C05360=1017.333,121.413,-117.741,166.979,53.925,159.921
C05361=1017.328,121.164,-117.723,166.976,53.934,159.922
C05362=1017.323,120.915,-117.704,166.972,53.942,159.923
C05363=1017.318,120.666,-117.685,166.969,53.951,159.924
C05364=1017.314,120.417,-117.667,166.966,53.960,159.926
C05365=1017.309,120.168,-117.648,166.963,53.969,159.927
C05366=1017.303,119.918,-117.630,166.960,53.978,159.928
C05367=1017.298,119.669,-117.612,166.957,53.987,159.929
C05368=1017.293,119.420,-117.593,166.954,53.996,159.930
C05369=1017.288,119.170,-117.575,166.951,54.005,159.931
C05370=1017.284,118.921,-117.557,166.948,54.014,159.932
C05371=1017.279,118.672,-117.538,166.945,54.023,159.934
C05372=1017.274,118.423,-117.520,166.942,54.031,159.934
C05373=1017.269,118.174,-117.501,166.939,54.040,159.936
C05374=1017.264,117.924,-117.483,166.937,54.049,159.937
C05375=1017.260,117.675,-117.465,166.934,54.058,159.938
C05376=1017.254,117.426,-117.446,166.931,54.067,159.939
C05377=1017.249,117.176,-117.428,166.928,54.076,159.940
C05378=1017.244,116.927,-117.409,166.925,54.085,159.941
C05379=1017.240,116.677,-117.391,166.922,54.094,159.943
C05380=1017.235,116.428,-117.373,166.919,54.103,159.944
C05381=1017.230,116.179,-117.354,166.916,54.111,159.945
C05382=1017.226,115.930,-117.335,166.913,54.120,159.946
C05383=1017.221,115.680,-117.317,166.911,54.129,159.947
C05384=1017.216,115.431,-117.299,166.907,54.137,159.948
C05385=1017.211,115.182,-117.281,166.904,54.147,159.949
C05386=1017.206,114.933,-117.262,166.902,54.156,159.950
C05387=1017.201,114.684,-117.244,166.899,54.165,159.952
C05388=1017.197,114.434,-117.226,166.895,54.173,159.953
C05389=1017.192,114.185,-117.208,166.892,54.182,159.954
C05390=1017.187,113.936,-117.189,166.890,54.191,159.955
C05391=1017.182,113.686,-117.171,166.887,54.199,159.956
C05392=1017.177,113.437,-117.153,166.884,54.208,159.957
C05393=1017.172,113.188,-117.134,166.881,54.218,159.958
C05394=1017.168,112.939,-117.116,166.878,54.227,159.960
C05395=1017.163,112.689,-117.098,166.875,54.235,159.960
C05396=1017.158,112.440,-117.080,166.873,54.244,159.962
C05397=1017.153,112.191,-117.062,166.870,54.253,159.963
C05398=1017.148,111.941,-117.043,166.867,54.261,159.964
C05399=1017.144,111.692,-117.025,166.864,54.270,159.965
C05400=1017.138,111.443,-117.008,166.861,54.280,159.966
C05401=1017.133,111.194,-116.990,166.858,54.289,159.967
C05402=1017.129,110.944,-116.971,166.855,54.298,159.969
C05403=1017.124,110.695,-116.953,166.852,54.307,159.970
C05404=1017.118,110.446,-116.936,166.849,54.315,159.971
C05405=1017.114,110.196,-116.918,166.846,54.324,159.972
C05406=1017.109,109.947,-116.900,166.843,54.334,159.973
C05407=1017.104,109.698,-116.883,166.842,54.342,159.974
C05408=1017.099,109.448,-116.864,166.839,54.351,159.976
C05409=1017.094,109.199,-116.846,166.835,54.360,159.977
C05410=1017.088,108.950,-116.829,166.832,54.369,159.978
C05411=1017.084,108.700,-116.810,166.830,54.378,159.979
C05412=1017.079,108.450,-116.793,166.827,54.387,159.980
C05413=1017.074,108.201,-116.775,166.824,54.396,159.981
C05414=1017.069,107.952,-116.757,166.821,54.406,159.982
C05415=1017.063,107.703,-116.740,166.818,54.415,159.984
C05416=1017.059,107.453,-116.722,166.815,54.424,159.985
C05417=1017.053,107.172,-116.702,166.812,54.434,159.986
C05418=1017.047,106.890,-116.682,166.808,54.444,159.987
C05419=1017.042,106.608,-116.662,166.805,54.455,159.989
C05420=1017.035,106.327,-116.642,166.803,54.464,159.990
C05421=1017.032,106.078,-116.625,166.800,54.474,159.991
C05422=1017.026,105.829,-116.607,166.797,54.483,159.993
C05423=1017.021,105.579,-116.589,166.794,54.491,159.993
C05424=1017.016,105.330,-116.572,166.791,54.500,159.995
C05425=1017.011,105.080,-116.554,166.788,54.509,159.996
C05426=1017.006,104.831,-116.537,166.785,54.519,159.997
C05427=1017.001,104.582,-116.518,166.782,54.528,159.998
C05428=1016.997,104.332,-116.501,166.780,54.537,159.999
C05429=1016.991,104.083,-116.483,166.776,54.545,160.000
C05430=1016.986,103.833,-116.465,166.773,54.555,160.002
C05431=1016.982,103.585,-116.449,166.772,54.563,160.003
C05432=1016.977,103.335,-116.431,166.769,54.573,160.004
C05433=1016.971,103.086,-116.413,166.766,54.582,160.005
C05434=1016.967,102.836,-116.396,166.763,54.591,160.006
C05435=1016.961,102.587,-116.378,166.760,54.599,160.007
C05436=1016.957,102.338,-116.360,166.757,54.608,160.009
C05437=1016.951,102.088,-116.343,166.754,54.618,160.010
C05438=1016.947,101.839,-116.325,166.751,54.627,160.011
C05439=1016.942,101.590,-116.308,166.749,54.635,160.012
C05440=1016.937,101.340,-116.290,166.746,54.644,160.013
C05441=1016.932,101.091,-116.272,166.744,54.653,160.014
C05442=1016.927,100.841,-116.255,166.741,54.662,160.016
C05443=1016.922,100.592,-116.237,166.738,54.672,160.017
C05444=1016.917,100.343,-116.220,166.735,54.680,160.018
C05445=1016.913,100.094,-116.202,166.732,54.689,160.019
C05446=1016.907,99.845,-116.185,166.730,54.698,160.020
C05447=1016.903,99.595,-116.167,166.727,54.707,160.021
C05448=1016.897,99.346,-116.150,166.724,54.716,160.022
C05449=1016.893,99.096,-116.132,166.721,54.725,160.024
C05450=1016.887,98.847,-116.115,166.718,54.734,160.025
C05451=1016.883,98.598,-116.098,166.716,54.743,160.026
C05452=1016.878,98.348,-116.080,166.713,54.752,160.027
C05453=1016.873,98.099,-116.063,166.710,54.761,160.028
C05454=1016.868,97.849,-116.046,166.707,54.770,160.029
C05455=1016.862,97.600,-116.029,166.704,54.779,160.031
C05456=1016.858,97.351,-116.012,166.701,54.789,160.032
C05457=1016.853,97.102,-115.994,166.700,54.797,160.033
C05458=1016.848,96.852,-115.977,166.697,54.807,160.034
C05459=1016.842,96.602,-115.961,166.694,54.816,160.035
C05460=1016.838,96.353,-115.942,166.691,54.825,160.037
C05461=1016.833,96.104,-115.926,166.688,54.833,160.038
C05462=1016.828,95.854,-115.909,166.685,54.843,160.039
C05463=1016.822,95.605,-115.892,166.683,54.852,160.040
C05464=1016.817,95.356,-115.875,166.680,54.861,160.041
C05465=1016.813,95.106,-115.858,166.677,54.870,160.042
C05466=1016.808,94.857,-115.840,166.674,54.880,160.044
C05467=1016.802,94.608,-115.823,166.671,54.888,160.045
C05468=1016.797,94.358,-115.806,166.669,54.897,160.046
C05469=1016.793,94.109,-115.789,166.667,54.906,160.047
C05470=1016.788,93.860,-115.772,166.664,54.915,160.048
C05471=1016.783,93.610,-115.755,166.661,54.925,160.050
C05472=1016.777,93.361,-115.737,166.658,54.933,160.050
C05473=1016.773,93.112,-115.720,166.655,54.942,160.052
C05474=1016.768,92.862,-115.703,166.652,54.951,160.053
C05475=1016.763,92.613,-115.686,166.650,54.961,160.054
C05476=1016.758,92.364,-115.669,166.647,54.970,160.055
C05477=1016.753,92.115,-115.652,166.645,54.978,160.056
C05478=1016.748,91.865,-115.635,166.642,54.987,160.058
C05479=1016.743,91.615,-115.618,166.639,54.997,160.059
C05480=1016.738,91.367,-115.601,166.637,55.006,160.060
C05481=1016.732,91.085,-115.582,166.633,55.015,160.061
C05482=1016.727,90.803,-115.562,166.631,55.025,160.063
C05483=1016.722,90.522,-115.543,166.627,55.036,160.064
C05484=1016.716,90.240,-115.524,166.624,55.046,160.065
C05485=1016.711,89.991,-115.507,166.621,55.055,160.066
C05486=1016.706,89.742,-115.490,166.619,55.063,160.067
C05487=1016.701,89.492,-115.473,166.616,55.073,160.069
C05488=1016.696,89.243,-115.456,166.614,55.082,160.070
C05489=1016.692,88.994,-115.439,166.611,55.091,160.071
C05490=1016.686,88.744,-115.422,166.608,55.100,160.072
C05491=1016.681,88.494,-115.406,166.605,55.109,160.073
C05492=1016.676,88.245,-115.389,166.602,55.118,160.074
C05493=1016.671,87.996,-115.372,166.600,55.127,160.076
C05494=1016.666,87.746,-115.355,166.597,55.137,160.077
C05495=1016.661,87.497,-115.339,166.594,55.146,160.078
C05496=1016.656,87.247,-115.322,166.593,55.155,160.079
C05497=1016.651,86.998,-115.305,166.590,55.163,160.080
C05498=1016.646,86.749,-115.289,166.587,55.173,160.082
C05499=1016.640,86.500,-115.272,166.584,55.182,160.083
C05500=1016.635,86.250,-115.256,166.581,55.191,160.084
C05501=1016.631,86.001,-115.239,166.579,55.200,160.085
C05502=1016.625,85.751,-115.222,166.576,55.210,160.086
C05503=1016.620,85.502,-115.205,166.573,55.218,160.087
C05504=1016.616,85.253,-115.189,166.570,55.228,160.089
C05505=1016.610,85.003,-115.172,166.568,55.237,160.090
C05506=1016.606,84.754,-115.156,166.565,55.246,160.091
C05507=1016.601,84.504,-115.139,166.562,55.255,160.092
C05508=1016.595,84.255,-115.122,166.560,55.263,160.093
C05509=1016.590,84.006,-115.106,166.557,55.273,160.095
C05510=1016.585,83.756,-115.089,166.555,55.282,160.096
C05511=1016.580,83.507,-115.073,166.552,55.291,160.097
C05512=1016.575,83.257,-115.057,166.550,55.301,160.098
C05513=1016.570,83.007,-115.040,166.546,55.309,160.099
C05514=1016.565,82.759,-115.023,166.544,55.318,160.100
C05515=1016.560,82.509,-115.006,166.541,55.328,160.102
C05516=1016.556,82.260,-114.990,166.539,55.337,160.103
C05517=1016.550,82.010,-114.973,166.536,55.345,160.104
C05518=1016.546,81.761,-114.957,166.534,55.354,160.105
C05519=1016.540,81.512,-114.940,166.531,55.364,160.106
C05520=1016.535,81.262,-114.923,166.528,55.372,160.107
C05521=1016.530,81.013,-114.908,166.525,55.382,160.109
C05522=1016.525,80.763,-114.891,166.523,55.391,160.110
C05523=1016.521,80.514,-114.874,166.521,55.400,160.111
C05524=1016.515,80.264,-114.857,166.518,55.408,160.112
C05525=1016.511,80.015,-114.841,166.515,55.418,160.113
C05526=1016.506,79.766,-114.824,166.513,55.427,160.115
C05527=1016.501,79.516,-114.808,166.509,55.436,160.116
C05528=1016.496,79.267,-114.792,166.507,55.445,160.117
C05529=1016.491,79.018,-114.776,166.505,55.454,160.118
C05530=1016.485,78.768,-114.759,166.502,55.462,160.119
C05531=1016.481,78.519,-114.742,166.499,55.472,160.120
C05532=1016.476,78.269,-114.726,166.497,55.481,160.122
C05533=1016.471,78.020,-114.710,166.494,55.490,160.123
C05534=1016.466,77.770,-114.693,166.492,55.499,160.124
C05535=1016.461,77.521,-114.676,166.489,55.507,160.125
C05536=1016.456,77.272,-114.659,166.486,55.516,160.126
C05537=1016.452,77.022,-114.644,166.484,55.526,160.127
C05538=1016.446,76.773,-114.627,166.481,55.534,160.128
C05539=1016.441,76.524,-114.611,166.478,55.544,160.130
C05540=1016.436,76.274,-114.595,166.477,55.553,160.131
C05541=1016.432,76.025,-114.578,166.474,55.562,160.132
C05542=1016.426,75.775,-114.562,166.471,55.570,160.133
C05543=1016.422,75.526,-114.546,166.468,55.580,160.134
C05544=1016.416,75.276,-114.530,166.466,55.589,160.136
C05545=1016.411,74.995,-114.512,166.463,55.600,160.137
C05546=1016.404,74.713,-114.494,166.460,55.610,160.138
C05547=1016.399,74.432,-114.475,166.457,55.619,160.139
C05548=1016.393,74.151,-114.457,166.454,55.630,160.141
C05549=1016.388,73.901,-114.441,166.451,55.639,160.142
C05550=1016.383,73.652,-114.425,166.449,55.649,160.143
C05551=1016.378,73.402,-114.409,166.445,55.657,160.144
C05552=1016.373,73.153,-114.393,166.444,55.666,160.146
C05553=1016.368,72.904,-114.377,166.441,55.675,160.147
C05554=1016.363,72.654,-114.361,166.438,55.684,160.148
C05555=1016.358,72.405,-114.345,166.436,55.693,160.149
C05556=1016.353,72.155,-114.329,166.433,55.703,160.150
C05557=1016.348,71.906,-114.312,166.430,55.711,160.151
C05558=1016.343,71.656,-114.297,166.428,55.721,160.152
C05559=1016.338,71.407,-114.280,166.426,55.730,160.154
C05560=1016.333,71.158,-114.265,166.423,55.738,160.155
C05561=1016.328,70.908,-114.248,166.420,55.748,160.156
C05562=1016.323,70.659,-114.232,166.418,55.757,160.157
C05563=1016.318,70.409,-114.216,166.415,55.766,160.158
C05564=1016.313,70.160,-114.200,166.412,55.775,160.159
C05565=1016.308,69.911,-114.185,166.411,55.784,160.161
C05566=1016.303,69.661,-114.168,166.408,55.793,160.162
C05567=1016.298,69.412,-114.153,166.405,55.802,160.163
C05568=1016.293,69.162,-114.136,166.403,55.811,160.164
C05569=1016.288,68.912,-114.120,166.399,55.820,160.165
C05570=1016.283,68.664,-114.104,166.397,55.829,160.167
C05571=1016.278,68.414,-114.088,166.395,55.837,160.168
C05572=1016.273,68.164,-114.073,166.392,55.847,160.169
C05573=1016.269,67.915,-114.057,166.390,55.856,160.170
C05574=1016.263,67.665,-114.041,166.387,55.865,160.171
C05575=1016.259,67.416,-114.025,166.384,55.874,160.172
C05576=1016.253,67.167,-114.009,166.382,55.884,160.174
C05577=1016.248,66.917,-113.994,166.380,55.892,160.175
C05578=1016.243,66.668,-113.978,166.377,55.901,160.176
C05579=1016.237,66.418,-113.962,166.375,55.911,160.177
C05580=1016.233,66.169,-113.946,166.372,55.919,160.178
C05581=1016.228,65.919,-113.931,166.369,55.929,160.179
C05582=1016.222,65.670,-113.915,166.367,55.938,160.181
C05583=1016.218,65.420,-113.899,166.364,55.947,160.182
C05584=1016.213,65.171,-113.884,166.362,55.956,160.183
C05585=1016.208,64.921,-113.868,166.359,55.964,160.184
C05586=1016.202,64.672,-113.852,166.357,55.974,160.185
C05587=1016.197,64.423,-113.837,166.354,55.983,160.187
C05588=1016.192,64.173,-113.820,166.351,55.992,160.188
C05589=1016.187,63.923,-113.805,166.349,56.001,160.189
C05590=1016.182,63.674,-113.790,166.346,56.011,160.190
C05591=1016.178,63.425,-113.774,166.344,56.019,160.191
C05592=1016.172,63.175,-113.758,166.342,56.028,160.192
C05593=1016.167,62.926,-113.743,166.339,56.037,160.193
C05594=1016.163,62.676,-113.727,166.336,56.046,160.195
C05595=1016.157,62.426,-113.712,166.334,56.056,160.196
C05596=1016.152,62.177,-113.696,166.331,56.064,160.197
C05597=1016.147,61.928,-113.681,166.328,56.074,160.198
C05598=1016.141,61.678,-113.666,166.326,56.083,160.199
C05599=1016.136,61.429,-113.651,166.323,56.093,160.201
C05600=1016.131,61.179,-113.635,166.320,56.101,160.202
C05601=1016.126,60.930,-113.620,166.318,56.111,160.203
C05602=1016.121,60.680,-113.605,166.316,56.120,160.204
C05603=1016.116,60.431,-113.589,166.314,56.129,160.206
C05604=1016.111,60.182,-113.574,166.311,56.138,160.206
C05605=1016.105,59.932,-113.559,166.308,56.147,160.208
C05606=1016.100,59.682,-113.544,166.306,56.157,160.209
C05607=1016.096,59.433,-113.528,166.303,56.166,160.210
C05608=1016.090,59.184,-113.513,166.300,56.175,160.211
C05609=1016.084,58.903,-113.496,166.298,56.185,160.213
C05610=1016.079,58.621,-113.479,166.295,56.196,160.214
C05611=1016.073,58.340,-113.461,166.293,56.206,160.215
C05612=1016.067,58.058,-113.444,166.289,56.216,160.217
C05613=1016.062,57.808,-113.429,166.287,56.225,160.218
C05614=1016.057,57.559,-113.413,166.284,56.235,160.219
C05615=1016.052,57.310,-113.398,166.281,56.243,160.220
C05616=1016.047,57.060,-113.383,166.279,56.253,160.221
C05617=1016.042,56.811,-113.368,166.276,56.262,160.223
C05618=1016.036,56.561,-113.352,166.273,56.271,160.224
C05619=1016.031,56.312,-113.337,166.272,56.280,160.225
C05620=1016.026,56.063,-113.322,166.269,56.289,160.226
C05621=1016.021,55.813,-113.307,166.267,56.298,160.227
C05622=1016.016,55.563,-113.292,166.264,56.307,160.228
C05623=1016.010,55.314,-113.277,166.261,56.316,160.229
C05624=1016.005,55.064,-113.262,166.259,56.326,160.231
C05625=1016.000,54.815,-113.246,166.256,56.334,160.232
C05626=1015.995,54.566,-113.231,166.253,56.344,160.233
C05627=1015.990,54.316,-113.216,166.252,56.352,160.234
C05628=1015.985,54.067,-113.201,166.249,56.361,160.235
C05629=1015.980,53.817,-113.186,166.246,56.370,160.236
C05630=1015.975,53.567,-113.171,166.244,56.380,160.238
C05631=1015.970,53.318,-113.156,166.241,56.388,160.239
C05632=1015.965,53.069,-113.141,166.238,56.398,160.240
C05633=1015.960,52.820,-113.125,166.237,56.406,160.241
C05634=1015.955,52.570,-113.110,166.234,56.416,160.242
C05635=1015.950,52.320,-113.096,166.231,56.424,160.243
C05636=1015.945,52.070,-113.080,166.229,56.434,160.245
C05637=1015.940,51.821,-113.064,166.226,56.442,160.246
C05638=1015.935,51.572,-113.049,166.225,56.452,160.247
C05639=1015.930,51.322,-113.034,166.222,56.460,160.248
C05640=1015.925,51.072,-113.020,166.219,56.470,160.249
C05641=1015.920,50.823,-113.004,166.216,56.478,160.250
C05642=1015.915,50.574,-112.989,166.214,56.488,160.252
C05643=1015.910,50.325,-112.974,166.212,56.496,160.253
C05644=1015.905,50.074,-112.959,166.209,56.505,160.254
C05645=1015.900,49.825,-112.944,166.207,56.514,160.255
C05646=1015.895,49.575,-112.929,166.204,56.523,160.256
C05647=1015.889,49.326,-112.914,166.201,56.533,160.257
C05648=1015.885,49.076,-112.899,166.200,56.541,160.258
C05649=1015.880,48.827,-112.884,166.197,56.550,160.259
C05650=1015.875,48.578,-112.869,166.194,56.559,160.261
C05651=1015.870,48.329,-112.854,166.191,56.568,160.262
C05652=1015.865,48.079,-112.839,166.189,56.576,160.263
C05653=1015.860,47.829,-112.824,166.187,56.586,160.264
C05654=1015.855,47.580,-112.809,166.184,56.594,160.265
C05655=1015.850,47.331,-112.794,166.181,56.603,160.266
C05656=1015.845,47.081,-112.779,166.180,56.612,160.268
C05657=1015.839,46.831,-112.764,166.177,56.621,160.268
C05658=1015.834,46.582,-112.749,166.174,56.630,160.269
C05659=1015.830,46.332,-112.734,166.171,56.639,160.270
C05660=1015.825,46.083,-112.719,166.170,56.648,160.272
C05661=1015.819,45.833,-112.704,166.167,56.656,160.273
C05662=1015.815,45.583,-112.689,166.164,56.665,160.274
C05663=1015.810,45.334,-112.674,166.163,56.674,160.275
C05664=1015.805,45.085,-112.659,166.160,56.683,160.276
C05665=1015.800,44.835,-112.645,166.157,56.692,160.277
C05666=1015.795,44.586,-112.629,166.154,56.701,160.278
C05667=1015.790,44.336,-112.614,166.152,56.709,160.280
C05668=1015.785,44.087,-112.600,166.150,56.718,160.281
C05669=1015.780,43.837,-112.585,166.147,56.727,160.282
C05670=1015.775,43.587,-112.570,166.145,56.736,160.283
C05671=1015.770,43.338,-112.555,166.143,56.744,160.284
C05672=1015.765,43.089,-112.540,166.140,56.753,160.285
C05673=1015.760,42.831,-112.524,166.138,56.762,160.286
C05674=1015.755,42.574,-112.509,166.135,56.771,160.287
C05675=1015.751,42.315,-112.494,166.133,56.780,160.289
C05676=1015.745,42.058,-112.479,166.130,56.789,160.290
C05677=1015.740,41.809,-112.464,166.127,56.798,160.291
C05678=1015.735,41.559,-112.449,166.125,56.807,160.292
C05679=1015.730,41.310,-112.435,166.122,56.816,160.293
C05680=1015.725,41.060,-112.420,166.120,56.825,160.294
C05681=1015.720,40.810,-112.406,166.118,56.834,160.295
C05682=1015.715,40.561,-112.390,166.115,56.843,160.296
C05683=1015.710,40.311,-112.377,166.112,56.852,160.297
C05684=1015.705,40.062,-112.361,166.111,56.861,160.299
C05685=1015.701,39.813,-112.347,166.108,56.870,160.300
C05686=1015.695,39.563,-112.333,166.105,56.878,160.301
C05687=1015.690,39.314,-112.318,166.103,56.887,160.302
C05688=1015.685,39.064,-112.304,166.101,56.896,160.303
C05689=1015.680,38.815,-112.289,166.099,56.905,160.304
C05690=1015.675,38.565,-112.275,166.096,56.914,160.305
C05691=1015.670,38.315,-112.260,166.093,56.923,160.306
C05692=1015.665,38.066,-112.245,166.092,56.932,160.308
C05693=1015.660,37.816,-112.231,166.089,56.941,160.309
C05694=1015.655,37.567,-112.217,166.086,56.949,160.310
C05695=1015.650,37.317,-112.202,166.083,56.958,160.311
C05696=1015.645,37.068,-112.187,166.081,56.967,160.312
C05697=1015.639,36.818,-112.173,166.079,56.976,160.313
C05698=1015.635,36.568,-112.159,166.076,56.985,160.314
C05699=1015.630,36.319,-112.144,166.074,56.993,160.316
C05700=1015.625,36.070,-112.130,166.072,57.002,160.317
C05701=1015.620,35.820,-112.116,166.069,57.012,160.318
C05702=1015.615,35.571,-112.102,166.067,57.020,160.319
C05703=1015.610,35.321,-112.087,166.064,57.029,160.320
C05704=1015.604,35.072,-112.073,166.061,57.038,160.321
C05705=1015.599,34.822,-112.058,166.060,57.047,160.322
C05706=1015.594,34.572,-112.044,166.057,57.056,160.323
C05707=1015.589,34.322,-112.030,166.054,57.065,160.324
C05708=1015.584,34.073,-112.017,166.051,57.074,160.325
C05709=1015.580,33.824,-112.002,166.049,57.083,160.327
C05710=1015.574,33.574,-111.988,166.047,57.092,160.328
C05711=1015.569,33.325,-111.973,166.044,57.100,160.329
C05712=1015.564,33.075,-111.959,166.042,57.109,160.330
C05713=1015.558,32.826,-111.945,166.039,57.119,160.331
C05714=1015.553,32.576,-111.931,166.038,57.127,160.332
C05715=1015.548,32.327,-111.917,166.035,57.136,160.333
C05716=1015.544,32.077,-111.903,166.032,57.145,160.334
C05717=1015.538,31.827,-111.889,166.029,57.154,160.335
C05718=1015.533,31.577,-111.875,166.028,57.163,160.337
C05719=1015.528,31.328,-111.861,166.025,57.172,160.338
C05720=1015.523,31.078,-111.846,166.023,57.181,160.339
C05721=1015.518,30.829,-111.833,166.020,57.189,160.340
C05722=1015.513,30.580,-111.818,166.018,57.198,160.341
C05723=1015.508,30.330,-111.804,166.015,57.207,160.342
C05724=1015.503,30.080,-111.789,166.012,57.215,160.343
C05725=1015.498,29.807,-111.774,166.010,57.225,160.345
C05726=1015.492,29.534,-111.759,166.007,57.235,160.346
C05727=1015.487,29.260,-111.744,166.005,57.245,160.347
C05728=1015.481,28.987,-111.729,166.003,57.254,160.348
C05729=1015.476,28.737,-111.714,166.000,57.263,160.349
C05730=1015.471,28.488,-111.701,165.997,57.272,160.350
C05731=1015.467,28.238,-111.686,165.995,57.280,160.352
C05732=1015.461,27.989,-111.672,165.993,57.289,160.353
C05733=1015.456,27.739,-111.658,165.990,57.298,160.354
C05734=1015.451,27.490,-111.644,165.988,57.306,160.355
C05735=1015.446,27.240,-111.630,165.985,57.315,160.356
C05736=1015.441,26.990,-111.616,165.983,57.324,160.357
C05737=1015.436,26.710,-111.600,165.980,57.334,160.358
C05738=1015.429,26.428,-111.585,165.977,57.344,160.359
C05739=1015.423,26.147,-111.569,165.975,57.355,160.361
C05740=1015.418,25.866,-111.554,165.972,57.364,160.362
C05741=1015.413,25.616,-111.540,165.970,57.373,160.363
C05742=1015.408,25.366,-111.525,165.967,57.382,160.364
C05743=1015.403,25.116,-111.512,165.965,57.390,160.365
C05744=1015.398,24.867,-111.499,165.962,57.399,160.366
C05745=1015.392,24.618,-111.485,165.960,57.408,160.367
C05746=1015.388,24.368,-111.470,165.957,57.417,160.368
C05747=1015.383,24.119,-111.457,165.955,57.425,160.369
C05748=1015.378,23.869,-111.444,165.953,57.434,160.370
C05749=1015.372,23.619,-111.430,165.950,57.443,160.371
C05750=1015.367,23.370,-111.416,165.947,57.452,160.373
C05751=1015.363,23.120,-111.402,165.945,57.460,160.374
C05752=1015.357,22.871,-111.388,165.943,57.469,160.375
C05753=1015.352,22.621,-111.375,165.940,57.478,160.376
C05754=1015.347,22.372,-111.361,165.938,57.487,160.377
C05755=1015.342,22.122,-111.348,165.935,57.495,160.378
C05756=1015.337,21.872,-111.334,165.933,57.504,160.379
C05757=1015.332,21.623,-111.320,165.930,57.513,160.380
C05758=1015.327,21.373,-111.307,165.928,57.522,160.381
C05759=1015.321,21.124,-111.293,165.926,57.531,160.382
C05760=1015.317,20.874,-111.280,165.923,57.539,160.383
C05761=1015.312,20.624,-111.265,165.921,57.548,160.385
C05762=1015.307,20.375,-111.252,165.919,57.557,160.386
C05763=1015.302,20.125,-111.239,165.916,57.566,160.387
C05764=1015.297,19.876,-111.225,165.914,57.574,160.388
C05765=1015.291,19.626,-111.211,165.912,57.583,160.389
C05766=1015.287,19.377,-111.197,165.908,57.591,160.390
C05767=1015.282,19.127,-111.184,165.907,57.600,160.391
C05768=1015.277,18.878,-111.170,165.904,57.609,160.392
C05769=1015.272,18.628,-111.157,165.901,57.617,160.393
C05770=1015.266,18.378,-111.143,165.900,57.626,160.394
C05771=1015.261,18.129,-111.130,165.897,57.635,160.395
C05772=1015.256,17.879,-111.117,165.894,57.644,160.396
C05773=1015.251,17.630,-111.103,165.893,57.652,160.397
C05774=1015.246,17.380,-111.090,165.890,57.661,160.398
C05775=1015.241,17.130,-111.076,165.887,57.670,160.399
C05776=1015.236,16.881,-111.063,165.884,57.679,160.400
C05777=1015.231,16.631,-111.049,165.882,57.687,160.401
C05778=1015.227,16.381,-111.036,165.880,57.696,160.402
C05779=1015.221,16.132,-111.022,165.877,57.704,160.403
C05780=1015.216,15.882,-111.008,165.875,57.713,160.405
C05781=1015.211,15.633,-110.996,165.873,57.722,160.406
C05782=1015.206,15.383,-110.982,165.870,57.731,160.407
C05783=1015.201,15.134,-110.969,165.868,57.739,160.408
C05784=1015.196,14.884,-110.955,165.865,57.747,160.409
C05785=1015.191,14.635,-110.942,165.863,57.756,160.410
C05786=1015.186,14.385,-110.928,165.861,57.765,160.411
C05787=1015.181,14.135,-110.915,165.858,57.774,160.412
C05788=1015.176,13.886,-110.902,165.856,57.781,160.413
C05789=1015.170,13.636,-110.889,165.853,57.790,160.414
C05790=1015.166,13.386,-110.876,165.850,57.799,160.415
C05791=1015.160,13.137,-110.862,165.849,57.808,160.416
C05792=1015.156,12.887,-110.849,165.846,57.817,160.417
C05793=1015.151,12.637,-110.836,165.844,57.826,160.418
C05794=1015.145,12.388,-110.822,165.841,57.833,160.419
C05795=1015.140,12.138,-110.810,165.839,57.842,160.420
C05796=1015.135,11.888,-110.797,165.836,57.851,160.421
C05797=1015.130,11.639,-110.783,165.833,57.860,160.422
C05798=1015.125,11.389,-110.770,165.832,57.869,160.424
C05799=1015.119,11.140,-110.758,165.829,57.878,160.425
C05800=1015.114,10.890,-110.745,165.827,57.887,160.426
C05801=1015.108,10.610,-110.730,165.825,57.896,160.427
C05802=1015.103,10.331,-110.715,165.821,57.906,160.428
C05803=1015.097,10.051,-110.702,165.819,57.915,160.429
C05804=1015.091,9.771,-110.687,165.816,57.925,160.430
C05805=1015.086,9.521,-110.673,165.813,57.934,160.431
C05806=1015.082,9.272,-110.661,165.811,57.942,160.432
C05807=1015.076,9.022,-110.647,165.808,57.951,160.433
C05808=1015.071,8.773,-110.635,165.806,57.960,160.434
C05809=1015.066,8.523,-110.621,165.804,57.968,160.436
C05810=1015.061,8.273,-110.609,165.801,57.977,160.436
C05811=1015.056,8.024,-110.596,165.798,57.986,160.437
C05812=1015.050,7.774,-110.583,165.797,57.994,160.439
C05813=1015.046,7.525,-110.570,165.794,58.003,160.440
C05814=1015.041,7.275,-110.557,165.791,58.011,160.440
C05815=1015.035,7.026,-110.544,165.789,58.020,160.442
C05816=1015.030,6.775,-110.531,165.787,58.029,160.443
C05817=1015.026,6.526,-110.519,165.784,58.037,160.444
C05818=1015.021,6.276,-110.506,165.782,58.046,160.445
C05819=1015.015,6.027,-110.492,165.779,58.054,160.446
C05820=1015.010,5.778,-110.480,165.777,58.062,160.447
C05821=1015.005,5.527,-110.467,165.774,58.071,160.448
C05822=1015.001,5.278,-110.454,165.773,58.080,160.449
C05823=1014.995,5.028,-110.441,165.770,58.088,160.450
C05824=1014.990,4.779,-110.428,165.767,58.097,160.451
C05825=1014.986,4.529,-110.416,165.765,58.105,160.452
C05826=1014.980,4.279,-110.402,165.762,58.114,160.453
C05827=1014.975,4.030,-110.390,165.761,58.122,160.454
C05828=1014.970,3.781,-110.377,165.758,58.130,160.455
C05829=1014.965,3.531,-110.364,165.755,58.139,160.456
C05830=1014.960,3.281,-110.351,165.753,58.147,160.457
C05831=1014.955,3.031,-110.338,165.750,58.156,160.458
C05832=1014.950,2.782,-110.326,165.748,58.164,160.459
C05833=1014.945,2.532,-110.313,165.746,58.173,160.460
C05834=1014.940,2.282,-110.300,165.743,58.181,160.461
C05835=1014.935,2.033,-110.287,165.741,58.190,160.462
C05836=1014.930,1.783,-110.275,165.739,58.198,160.463
C05837=1014.925,1.533,-110.261,165.736,58.206,160.464
C05838=1014.920,1.284,-110.249,165.734,58.214,160.465
C05839=1014.915,1.035,-110.237,165.731,58.223,160.465
C05840=1014.910,0.784,-110.223,165.729,58.231,160.467
C05841=1014.906,0.535,-110.211,165.726,58.239,160.467
C05842=1014.900,0.286,-110.198,165.725,58.248,160.469
C05843=1014.895,0.035,-110.185,165.722,58.256,160.469
C05844=1014.890,-0.214,-110.172,165.719,58.264,160.470
C05845=1014.886,-0.464,-110.160,165.717,58.273,160.471
C05846=1014.880,-0.713,-110.147,165.715,58.281,160.472
C05847=1014.875,-0.963,-110.134,165.712,58.290,160.473
C05848=1014.871,-1.212,-110.122,165.710,58.298,160.474
C05849=1014.866,-1.462,-110.109,165.707,58.306,160.475
C05850=1014.860,-1.712,-110.096,165.705,58.314,160.476
C05851=1014.856,-1.961,-110.083,165.702,58.323,160.477
C05852=1014.851,-2.211,-110.071,165.700,58.330,160.478
C05853=1014.845,-2.461,-110.058,165.697,58.339,160.479
C05854=1014.841,-2.710,-110.045,165.695,58.347,160.480
C05855=1014.836,-2.960,-110.033,165.693,58.355,160.481
C05856=1014.832,-3.209,-110.020,165.690,58.363,160.482
C05857=1014.826,-3.459,-110.007,165.688,58.371,160.483
C05858=1014.821,-3.708,-109.994,165.686,58.380,160.484
C05859=1014.817,-3.958,-109.982,165.683,58.388,160.485
C05860=1014.812,-4.207,-109.969,165.680,58.396,160.485
C05861=1014.806,-4.458,-109.957,165.678,58.404,160.486
C05862=1014.802,-4.707,-109.944,165.677,58.413,160.487
C05863=1014.797,-4.957,-109.932,165.674,58.421,160.488
C05864=1014.792,-5.206,-109.919,165.670,58.429,160.489
C05865=1014.786,-5.484,-109.906,165.669,58.439,160.490
C05866=1014.781,-5.762,-109.893,165.666,58.448,160.491
C05867=1014.775,-6.039,-109.879,165.663,58.457,160.492
C05868=1014.769,-6.317,-109.865,165.660,58.466,160.493
C05869=1014.764,-6.566,-109.854,165.658,58.475,160.495
C05870=1014.759,-6.817,-109.840,165.655,58.483,160.495
C05871=1014.754,-7.066,-109.828,165.653,58.491,160.496
C05872=1014.749,-7.316,-109.817,165.651,58.500,160.497
C05873=1014.744,-7.565,-109.804,165.649,58.508,160.498
C05874=1014.739,-7.815,-109.793,165.646,58.516,160.499
C05875=1014.733,-8.065,-109.780,165.644,58.525,160.500
C05876=1014.729,-8.314,-109.767,165.641,58.533,160.501
C05877=1014.724,-8.564,-109.756,165.639,58.541,160.502
C05878=1014.718,-8.813,-109.744,165.636,58.549,160.503
C05879=1014.714,-9.063,-109.731,165.634,58.558,160.504
C05880=1014.709,-9.313,-109.719,165.631,58.566,160.505
C05881=1014.704,-9.563,-109.706,165.629,58.574,160.506
C05882=1014.699,-9.813,-109.695,165.626,58.582,160.506
C05883=1014.693,-10.062,-109.682,165.625,58.591,160.508
C05884=1014.689,-10.312,-109.670,165.621,58.599,160.508
C05885=1014.684,-10.561,-109.658,165.619,58.607,160.509
C05886=1014.678,-10.810,-109.646,165.616,58.615,160.510
C05887=1014.674,-11.060,-109.634,165.614,58.623,160.511
C05888=1014.668,-11.310,-109.621,165.612,58.631,160.512
C05889=1014.663,-11.560,-109.610,165.610,58.640,160.513
C05890=1014.659,-11.810,-109.597,165.608,58.648,160.514
C05891=1014.654,-12.059,-109.586,165.605,58.656,160.515
C05892=1014.648,-12.309,-109.573,165.602,58.664,160.516
C05893=1014.644,-12.559,-109.561,165.600,58.672,160.517
C05894=1014.639,-12.808,-109.549,165.597,58.680,160.518
C05895=1014.634,-13.058,-109.538,165.595,58.688,160.518
C05896=1014.629,-13.307,-109.525,165.592,58.696,160.519
C05897=1014.624,-13.557,-109.513,165.590,58.704,160.520
C05898=1014.619,-13.806,-109.501,165.588,58.712,160.521
C05899=1014.614,-14.057,-109.489,165.585,58.720,160.522
C05900=1014.609,-14.306,-109.477,165.583,58.728,160.523
C05901=1014.604,-14.556,-109.465,165.581,58.736,160.524
C05902=1014.599,-14.805,-109.452,165.578,58.744,160.525
C05903=1014.594,-15.055,-109.441,165.576,58.752,160.526
C05904=1014.589,-15.305,-109.429,165.574,58.760,160.526
C05905=1014.585,-15.554,-109.417,165.571,58.768,160.527
C05906=1014.580,-15.804,-109.405,165.569,58.776,160.528
C05907=1014.575,-16.054,-109.392,165.567,58.784,160.529
C05908=1014.570,-16.304,-109.381,165.564,58.792,160.530
C05909=1014.565,-16.553,-109.370,165.562,58.800,160.531
C05910=1014.560,-16.803,-109.358,165.559,58.809,160.532
C05911=1014.555,-17.052,-109.346,165.557,58.817,160.533
C05912=1014.550,-17.302,-109.334,165.553,58.825,160.533
C05913=1014.545,-17.552,-109.323,165.551,58.833,160.534
C05914=1014.540,-17.802,-109.311,165.549,58.841,160.535
C05915=1014.534,-18.051,-109.299,165.546,58.849,160.536
C05916=1014.529,-18.301,-109.288,165.544,58.857,160.537
C05917=1014.524,-18.551,-109.276,165.541,58.865,160.538
C05918=1014.519,-18.800,-109.265,165.539,58.873,160.539
C05919=1014.515,-19.050,-109.252,165.537,58.881,160.540
C05920=1014.510,-19.300,-109.241,165.534,58.889,160.540
C05921=1014.505,-19.549,-109.229,165.532,58.897,160.541
C05922=1014.500,-19.799,-109.218,165.530,58.905,160.542
C05923=1014.495,-20.049,-109.206,165.527,58.913,160.543
C05924=1014.489,-20.298,-109.194,165.525,58.921,160.544
C05925=1014.484,-20.548,-109.182,165.523,58.929,160.545
C05926=1014.479,-20.798,-109.171,165.520,58.937,160.546
C05927=1014.474,-21.048,-109.160,165.518,58.945,160.547
C05928=1014.469,-21.297,-109.148,165.516,58.953,160.548
C05929=1014.464,-21.573,-109.135,165.513,58.962,160.548
C05930=1014.458,-21.849,-109.122,165.511,58.971,160.550
C05931=1014.453,-22.125,-109.109,165.508,58.979,160.550
C05932=1014.448,-22.401,-109.097,165.505,58.988,160.551
C05933=1014.443,-22.651,-109.085,165.502,58.996,160.552
C05934=1014.438,-22.900,-109.073,165.499,59.004,160.553
C05935=1014.433,-23.150,-109.062,165.498,59.011,160.554
C05936=1014.428,-23.399,-109.050,165.496,59.019,160.555
C05937=1014.423,-23.649,-109.039,165.492,59.028,160.555
C05938=1014.418,-23.899,-109.027,165.490,59.035,160.556
C05939=1014.413,-24.148,-109.016,165.488,59.043,160.557
C05940=1014.408,-24.398,-109.005,165.486,59.051,160.558
C05941=1014.403,-24.648,-108.993,165.483,59.059,160.559
C05942=1014.398,-24.897,-108.982,165.480,59.066,160.559
C05943=1014.393,-25.147,-108.970,165.478,59.074,160.560
C05944=1014.388,-25.397,-108.959,165.476,59.082,160.561
C05945=1014.383,-25.647,-108.947,165.473,59.090,160.562
C05946=1014.378,-25.897,-108.936,165.471,59.097,160.563
C05947=1014.374,-26.146,-108.925,165.469,59.105,160.564
C05948=1014.369,-26.395,-108.912,165.466,59.113,160.564
C05949=1014.364,-26.645,-108.900,165.464,59.120,160.565
C05950=1014.359,-26.895,-108.889,165.462,59.128,160.566
C05951=1014.354,-27.145,-108.878,165.459,59.136,160.567
C05952=1014.349,-27.394,-108.866,165.456,59.143,160.567
C05953=1014.345,-27.644,-108.855,165.454,59.151,160.568
C05954=1014.340,-27.894,-108.844,165.452,59.159,160.569
C05955=1014.335,-28.144,-108.833,165.449,59.166,160.570
C05956=1014.329,-28.393,-108.822,165.446,59.175,160.571
C05957=1014.324,-28.643,-108.810,165.445,59.182,160.572
C05958=1014.319,-28.893,-108.799,165.442,59.190,160.572
C05959=1014.315,-29.142,-108.788,165.440,59.198,160.573
C05960=1014.310,-29.392,-108.778,165.437,59.206,160.574
C05961=1014.305,-29.642,-108.766,165.434,59.213,160.575
C05962=1014.300,-29.892,-108.755,165.432,59.221,160.576
C05963=1014.295,-30.141,-108.743,165.431,59.229,160.577
C05964=1014.290,-30.391,-108.732,165.427,59.237,160.577
C05965=1014.285,-30.641,-108.722,165.425,59.244,160.578
C05966=1014.280,-30.890,-108.710,165.422,59.252,160.579
C05967=1014.275,-31.140,-108.699,165.420,59.260,160.580
C05968=1014.270,-31.389,-108.688,165.417,59.268,160.580
C05969=1014.265,-31.640,-108.678,165.415,59.275,160.581
C05970=1014.260,-31.889,-108.666,165.413,59.283,160.582
C05971=1014.255,-32.139,-108.655,165.410,59.290,160.583
C05972=1014.251,-32.388,-108.644,165.408,59.298,160.584
C05973=1014.245,-32.638,-108.634,165.406,59.305,160.584
C05974=1014.240,-32.888,-108.622,165.403,59.314,160.585
C05975=1014.236,-33.137,-108.611,165.400,59.321,160.586
C05976=1014.231,-33.388,-108.600,165.398,59.329,160.587
C05977=1014.225,-33.637,-108.589,165.396,59.336,160.587
C05978=1014.220,-33.887,-108.578,165.393,59.343,160.588
C05979=1014.216,-34.136,-108.567,165.391,59.351,160.589
C05980=1014.211,-34.386,-108.556,165.389,59.358,160.590
C05981=1014.205,-34.636,-108.545,165.387,59.366,160.591
C05982=1014.201,-34.885,-108.534,165.383,59.374,160.591
C05983=1014.196,-35.135,-108.523,165.381,59.381,160.592
C05984=1014.191,-35.385,-108.512,165.379,59.389,160.593
C05985=1014.186,-35.634,-108.501,165.376,59.396,160.593
C05986=1014.182,-35.884,-108.490,165.374,59.404,160.594
C05987=1014.177,-36.134,-108.479,165.372,59.411,160.595
C05988=1014.172,-36.384,-108.469,165.369,59.419,160.596
C05989=1014.167,-36.633,-108.458,165.367,59.426,160.596
C05990=1014.162,-36.883,-108.446,165.365,59.434,160.597
C05991=1014.158,-37.133,-108.436,165.362,59.441,160.598
C05992=1014.153,-37.383,-108.424,165.360,59.448,160.599
C05993=1014.147,-37.657,-108.412,165.357,59.457,160.599
C05994=1014.142,-37.932,-108.400,165.355,59.465,160.600
C05995=1014.137,-38.208,-108.388,165.352,59.473,160.601
C05996=1014.131,-38.482,-108.377,165.348,59.481,160.601
C05997=1014.126,-38.731,-108.366,165.347,59.488,160.603
C05998=1014.121,-38.982,-108.355,165.345,59.495,160.603
C05999=1014.116,-39.231,-108.344,165.342,59.503,160.604
C06000=1014.112,-39.481,-108.334,165.340,59.510,160.605
C06001=1014.107,-39.731,-108.322,165.337,59.517,160.605
C06002=1014.103,-39.980,-108.312,165.334,59.525,160.606
C06003=1014.097,-40.230,-108.301,165.332,59.533,160.607
C06004=1014.091,-40.480,-108.291,165.329,59.540,160.607
C06005=1014.087,-40.730,-108.281,165.327,59.547,160.608
C06006=1014.081,-40.979,-108.270,165.325,59.555,160.609
C06007=1014.077,-41.229,-108.259,165.322,59.562,160.610
C06008=1014.072,-41.479,-108.249,165.320,59.569,160.610
C06009=1014.068,-41.728,-108.238,165.317,59.577,160.611
C06010=1014.062,-41.978,-108.228,165.315,59.585,160.612
C06011=1014.058,-42.227,-108.217,165.313,59.592,160.613
C06012=1014.052,-42.477,-108.207,165.310,59.599,160.613
C06013=1014.048,-42.728,-108.196,165.308,59.606,160.614
C06014=1014.042,-42.977,-108.185,165.305,59.613,160.615
C06015=1014.038,-43.227,-108.175,165.303,59.621,160.615
C06016=1014.033,-43.476,-108.165,165.300,59.628,160.616
///RCONF 1,0,0,1,0,0,0,0,0,0,0,0,0,0,0,0,0,0,0,0,0,0,0,0
C06017=1014.028,-43.727,-108.154,165.298,59.636,160.617
C06018=1014.023,-43.976,-108.143,165.296,59.643,160.618
C06019=1014.018,-44.226,-108.133,165.293,59.650,160.618
C06020=1014.014,-44.475,-108.123,165.291,59.658,160.619
C06021=1014.008,-44.725,-108.112,165.288,59.665,160.619
C06022=1014.004,-44.975,-108.102,165.286,59.672,160.620
C06023=1013.998,-45.225,-108.091,165.283,59.679,160.621
C06024=1013.994,-45.474,-108.081,165.282,59.686,160.622
C06025=1013.988,-45.724,-108.070,165.279,59.693,160.622
C06026=1013.984,-45.974,-108.060,165.277,59.700,160.623
C06027=1013.979,-46.224,-108.050,165.274,59.708,160.624
C06028=1013.975,-46.473,-108.039,165.272,59.715,160.624
C06029=1013.970,-46.722,-108.029,165.269,59.722,160.625
C06030=1013.965,-46.973,-108.018,165.267,59.729,160.626
C06031=1013.960,-47.222,-108.008,165.263,59.736,160.626
C06032=1013.956,-47.473,-107.997,165.262,59.743,160.627
C06033=1013.951,-47.722,-107.988,165.259,59.750,160.627
C06034=1013.945,-47.971,-107.977,165.257,59.757,160.628
C06035=1013.941,-48.221,-107.966,165.254,59.764,160.629
C06036=1013.935,-48.471,-107.956,165.252,59.772,160.629
C06037=1013.931,-48.721,-107.946,165.249,59.779,160.630
C06038=1013.926,-48.970,-107.936,165.247,59.785,160.631
C06039=1013.921,-49.220,-107.925,165.245,59.792,160.631
C06040=1013.917,-49.470,-107.915,165.242,59.799,160.632
C06041=1013.912,-49.720,-107.904,165.240,59.807,160.633
C06042=1013.907,-49.969,-107.894,165.237,59.814,160.633
C06043=1013.903,-50.219,-107.884,165.235,59.820,160.634
C06044=1013.898,-50.469,-107.874,165.233,59.827,160.634
C06045=1013.893,-50.719,-107.863,165.230,59.834,160.635
C06046=1013.888,-50.969,-107.853,165.227,59.841,160.635
C06047=1013.884,-51.219,-107.843,165.226,59.848,160.636
C06048=1013.879,-51.469,-107.833,165.223,59.855,160.637
C06049=1013.874,-51.718,-107.823,165.221,59.862,160.638
C06050=1013.869,-51.968,-107.813,165.218,59.869,160.638
C06051=1013.863,-52.218,-107.803,165.216,59.877,160.639
C06052=1013.859,-52.467,-107.793,165.213,59.884,160.639
C06053=1013.854,-52.717,-107.783,165.211,59.891,160.640
C06054=1013.849,-52.967,-107.774,165.208,59.898,160.640
C06055=1013.844,-53.217,-107.764,165.206,59.904,160.641
C06056=1013.839,-53.466,-107.754,165.204,59.912,160.642
C06057=1013.833,-53.741,-107.743,165.201,59.920,160.643
C06058=1013.828,-54.016,-107.732,165.198,59.927,160.643
C06059=1013.823,-54.291,-107.721,165.195,59.935,160.644
C06060=1013.817,-54.567,-107.711,165.193,59.943,160.645
C06061=1013.812,-54.817,-107.701,165.190,59.950,160.645
C06062=1013.807,-55.066,-107.691,165.187,59.957,160.646
C06063=1013.802,-55.315,-107.681,165.186,59.964,160.647
C06064=1013.797,-55.565,-107.672,165.183,59.971,160.647
C06065=1013.792,-55.816,-107.662,165.180,59.978,160.648
C06066=1013.787,-56.065,-107.652,165.178,59.985,160.648
C06067=1013.783,-56.314,-107.643,165.175,59.992,160.649
C06068=1013.777,-56.565,-107.632,165.173,59.998,160.649
C06069=1013.773,-56.815,-107.623,165.171,60.005,160.650
C06070=1013.768,-57.064,-107.614,165.168,60.013,160.651
C06071=1013.764,-57.314,-107.603,165.166,60.019,160.651
C06072=1013.758,-57.564,-107.593,165.164,60.026,160.652
C06073=1013.754,-57.814,-107.584,165.161,60.033,160.653
C06074=1013.749,-58.063,-107.574,165.158,60.040,160.653
C06075=1013.744,-58.313,-107.564,165.157,60.047,160.654
C06076=1013.740,-58.563,-107.555,165.154,60.053,160.654
C06077=1013.734,-58.813,-107.545,165.151,60.060,160.655
C06078=1013.729,-59.062,-107.535,165.149,60.066,160.655
C06079=1013.724,-59.312,-107.525,165.147,60.074,160.656
C06080=1013.720,-59.562,-107.516,165.144,60.080,160.656
C06081=1013.714,-59.812,-107.506,165.142,60.087,160.657
C06082=1013.710,-60.061,-107.496,165.139,60.094,160.658
C06083=1013.705,-60.311,-107.487,165.137,60.101,160.658
C06084=1013.700,-60.561,-107.478,165.135,60.107,160.659
C06085=1013.695,-60.810,-107.468,165.131,60.113,160.659
C06086=1013.691,-61.060,-107.459,165.130,60.120,160.660
C06087=1013.685,-61.310,-107.449,165.127,60.127,160.660
C06088=1013.681,-61.560,-107.439,165.126,60.134,160.661
C06089=1013.676,-61.810,-107.430,165.122,60.140,160.661
C06090=1013.671,-62.059,-107.420,165.119,60.147,160.662
C06091=1013.667,-62.309,-107.411,165.118,60.153,160.663
C06092=1013.662,-62.558,-107.401,165.115,60.160,160.663
C06093=1013.657,-62.809,-107.392,165.113,60.166,160.663
C06094=1013.652,-63.059,-107.382,165.110,60.173,160.664
C06095=1013.647,-63.308,-107.372,165.108,60.179,160.665
C06096=1013.643,-63.558,-107.363,165.105,60.186,160.665
C06097=1013.638,-63.807,-107.353,165.103,60.192,160.666
C06098=1013.633,-64.057,-107.344,165.101,60.199,160.666
C06099=1013.628,-64.307,-107.334,165.099,60.205,160.667
C06100=1013.624,-64.556,-107.324,165.095,60.212,160.667
C06101=1013.618,-64.807,-107.315,165.093,60.218,160.668
C06102=1013.614,-65.056,-107.305,165.090,60.224,160.668
C06103=1013.610,-65.307,-107.295,165.088,60.231,160.668
C06104=1013.605,-65.556,-107.286,165.086,60.238,160.669
C06105=1013.600,-65.806,-107.277,165.084,60.244,160.670
C06106=1013.596,-66.056,-107.267,165.082,60.250,160.670
C06107=1013.591,-66.306,-107.258,165.079,60.257,160.671
C06108=1013.586,-66.555,-107.248,165.077,60.263,160.671
C06109=1013.582,-66.805,-107.239,165.073,60.269,160.671
C06110=1013.577,-67.054,-107.229,165.071,60.275,160.672
C06111=1013.572,-67.304,-107.220,165.069,60.281,160.672
C06112=1013.568,-67.554,-107.210,165.066,60.288,160.673
C06113=1013.563,-67.804,-107.201,165.064,60.294,160.673
C06114=1013.558,-68.053,-107.191,165.062,60.300,160.674
C06115=1013.554,-68.303,-107.182,165.059,60.307,160.674
C06116=1013.549,-68.553,-107.173,165.057,60.313,160.675
C06117=1013.544,-68.803,-107.163,165.055,60.319,160.675
C06118=1013.539,-69.053,-107.154,165.052,60.325,160.676
C06119=1013.534,-69.303,-107.144,165.050,60.331,160.676
C06120=1013.530,-69.553,-107.135,165.048,60.337,160.677
C06121=1013.524,-69.828,-107.125,165.045,60.344,160.677
C06122=1013.520,-70.104,-107.114,165.042,60.351,160.678
C06123=1013.514,-70.380,-107.104,165.039,60.358,160.678
C06124=1013.510,-70.657,-107.094,165.037,60.364,160.678
C06125=1013.505,-70.906,-107.084,165.034,60.371,160.679
C06126=1013.500,-71.156,-107.075,165.032,60.377,160.679
C06127=1013.495,-71.406,-107.065,165.030,60.383,160.680
C06128=1013.491,-71.656,-107.056,165.028,60.389,160.680
C06129=1013.486,-71.906,-107.047,165.024,60.395,160.680
C06130=1013.481,-72.155,-107.037,165.022,60.401,160.681
C06131=1013.477,-72.405,-107.028,165.020,60.407,160.681
C06132=1013.472,-72.655,-107.019,165.018,60.413,160.682
C06133=1013.468,-72.905,-107.009,165.016,60.418,160.682
C06134=1013.463,-73.155,-107.000,165.014,60.424,160.683
C06135=1013.459,-73.404,-106.992,165.010,60.431,160.683
C06136=1013.454,-73.653,-106.982,165.008,60.436,160.683
C06137=1013.450,-73.903,-106.973,165.006,60.442,160.684
C06138=1013.445,-74.153,-106.964,165.004,60.448,160.684
C06139=1013.440,-74.403,-106.954,165.001,60.454,160.684
C06140=1013.436,-74.653,-106.945,164.999,60.460,160.685
C06141=1013.431,-74.903,-106.936,164.996,60.465,160.685
C06142=1013.427,-75.153,-106.927,164.993,60.472,160.685
C06143=1013.422,-75.403,-106.918,164.991,60.478,160.686
C06144=1013.417,-75.653,-106.909,164.989,60.484,160.687
C06145=1013.412,-75.902,-106.899,164.987,60.489,160.687
C06146=1013.408,-76.151,-106.891,164.985,60.495,160.687
C06147=1013.403,-76.401,-106.882,164.981,60.502,160.688
C06148=1013.398,-76.651,-106.873,164.979,60.508,160.688
C06149=1013.394,-76.901,-106.864,164.977,60.513,160.688
C06150=1013.389,-77.151,-106.855,164.975,60.519,160.689
C06151=1013.384,-77.401,-106.846,164.972,60.525,160.689
C06152=1013.380,-77.651,-106.837,164.970,60.531,160.690
C06153=1013.375,-77.900,-106.829,164.968,60.537,160.690
C06154=1013.370,-78.150,-106.820,164.965,60.542,160.690
C06155=1013.366,-78.400,-106.811,164.962,60.549,160.691
C06156=1013.361,-78.650,-106.802,164.960,60.554,160.691
C06157=1013.356,-78.900,-106.793,164.958,60.560,160.691
C06158=1013.352,-79.149,-106.785,164.955,60.566,160.692
C06159=1013.347,-79.399,-106.776,164.953,60.572,160.692
C06160=1013.342,-79.649,-106.767,164.950,60.577,160.692
C06161=1013.338,-79.899,-106.758,164.948,60.583,160.693
C06162=1013.333,-80.149,-106.749,164.945,60.589,160.693
C06163=1013.328,-80.399,-106.740,164.944,60.595,160.694
C06164=1013.324,-80.649,-106.731,164.941,60.600,160.694
C06165=1013.319,-80.898,-106.723,164.939,60.606,160.694
C06166=1013.315,-81.148,-106.715,164.936,60.612,160.695
C06167=1013.309,-81.398,-106.706,164.934,60.618,160.695
C06168=1013.305,-81.648,-106.697,164.932,60.624,160.696
C06169=1013.300,-81.897,-106.689,164.929,60.629,160.696
C06170=1013.295,-82.147,-106.681,164.926,60.636,160.696
C06171=1013.291,-82.397,-106.672,164.924,60.641,160.696
C06172=1013.285,-82.647,-106.664,164.922,60.647,160.697
C06173=1013.282,-82.896,-106.655,164.919,60.653,160.697
C06174=1013.276,-83.146,-106.647,164.917,60.659,160.698
C06175=1013.272,-83.397,-106.638,164.914,60.664,160.698
C06176=1013.267,-83.646,-106.630,164.912,60.669,160.698
C06177=1013.262,-83.896,-106.622,164.910,60.676,160.698
C06178=1013.258,-84.146,-106.613,164.907,60.681,160.699
C06179=1013.253,-84.396,-106.605,164.905,60.687,160.699
C06180=1013.249,-84.645,-106.596,164.902,60.692,160.699
C06181=1013.243,-84.895,-106.588,164.900,60.698,160.700
C06182=1013.238,-85.145,-106.579,164.899,60.703,160.700
C06183=1013.235,-85.395,-106.571,164.896,60.709,160.701
C06184=1013.229,-85.644,-106.563,164.893,60.714,160.701
C06185=1013.225,-85.922,-106.553,164.890,60.721,160.701
C06186=1013.219,-86.200,-106.544,164.888,60.727,160.702
C06187=1013.214,-86.479,-106.535,164.885,60.733,160.701
C06188=1013.209,-86.756,-106.526,164.883,60.739,160.702
C06189=1013.205,-87.006,-106.517,164.880,60.744,160.702
C06190=1013.199,-87.256,-106.508,164.877,60.750,160.702
C06191=1013.195,-87.505,-106.501,164.875,60.756,160.703
C06192=1013.190,-87.755,-106.492,164.874,60.761,160.703
C06193=1013.185,-88.005,-106.483,164.871,60.766,160.704
C06194=1013.181,-88.255,-106.475,164.868,60.771,160.704
C06195=1013.176,-88.505,-106.467,164.866,60.777,160.704
C06196=1013.172,-88.754,-106.459,164.863,60.782,160.704
C06197=1013.167,-89.005,-106.450,164.861,60.787,160.705
C06198=1013.162,-89.254,-106.442,164.859,60.792,160.705
C06199=1013.158,-89.504,-106.434,164.856,60.798,160.705
C06200=1013.153,-89.754,-106.425,164.853,60.803,160.705
C06201=1013.149,-90.004,-106.418,164.852,60.808,160.706
C06202=1013.144,-90.254,-106.409,164.849,60.813,160.706
C06203=1013.139,-90.503,-106.400,164.846,60.819,160.706
C06204=1013.135,-90.753,-106.392,164.844,60.824,160.706
C06205=1013.130,-91.003,-106.384,164.842,60.829,160.706
C06206=1013.126,-91.253,-106.376,164.840,60.834,160.707
C06207=1013.121,-91.503,-106.367,164.837,60.840,160.707
C06208=1013.117,-91.752,-106.360,164.835,60.845,160.707
C06209=1013.112,-92.002,-106.351,164.833,60.850,160.707
C06210=1013.107,-92.253,-106.343,164.830,60.855,160.708
C06211=1013.104,-92.502,-106.334,164.828,60.860,160.708
C06212=1013.099,-92.752,-106.327,164.826,60.866,160.708
C06213=1013.094,-93.001,-106.318,164.823,60.870,160.708
C06214=1013.090,-93.252,-106.310,164.821,60.875,160.709
C06215=1013.085,-93.501,-106.302,164.818,60.881,160.709
C06216=1013.081,-93.752,-106.294,164.817,60.886,160.709
C06217=1013.076,-94.001,-106.286,164.813,60.890,160.709
C06218=1013.071,-94.251,-106.278,164.812,60.895,160.709
C06219=1013.067,-94.500,-106.269,164.809,60.900,160.710
C06220=1013.062,-94.751,-106.261,164.807,60.905,160.710
C06221=1013.058,-95.000,-106.253,164.804,60.910,160.710
C06222=1013.053,-95.250,-106.245,164.802,60.915,160.710
C06223=1013.049,-95.499,-106.237,164.800,60.920,160.710
C06224=1013.045,-95.750,-106.228,164.797,60.924,160.710
C06225=1013.040,-95.999,-106.220,164.795,60.930,160.711
C06226=1013.035,-96.249,-106.212,164.793,60.935,160.711
C06227=1013.031,-96.499,-106.204,164.790,60.939,160.711
C06228=1013.026,-96.749,-106.196,164.788,60.944,160.711
C06229=1013.022,-96.999,-106.188,164.785,60.949,160.711
C06230=1013.018,-97.248,-106.180,164.783,60.954,160.712
C06231=1013.013,-97.498,-106.172,164.781,60.958,160.712
C06232=1013.009,-97.748,-106.164,164.778,60.963,160.712
C06233=1013.004,-97.998,-106.156,164.776,60.968,160.712
C06234=1013.000,-98.247,-106.148,164.773,60.973,160.712
C06235=1012.995,-98.498,-106.140,164.772,60.978,160.712
C06236=1012.991,-98.748,-106.132,164.769,60.982,160.712
C06237=1012.986,-98.997,-106.124,164.767,60.987,160.713
C06238=1012.981,-99.247,-106.116,164.764,60.992,160.712
C06239=1012.977,-99.497,-106.109,164.762,60.997,160.713
C06240=1012.972,-99.747,-106.101,164.760,61.002,160.713
C06241=1012.968,-99.997,-106.094,164.757,61.006,160.713
C06242=1012.963,-100.247,-106.086,164.756,61.011,160.714
C06243=1012.959,-100.496,-106.077,164.752,61.016,160.713
C06244=1012.954,-100.746,-106.070,164.751,61.021,160.714
C06245=1012.949,-100.996,-106.062,164.748,61.025,160.714
C06246=1012.945,-101.246,-106.055,164.746,61.031,160.714
C06247=1012.941,-101.496,-106.047,164.743,61.035,160.714
C06248=1012.936,-101.746,-106.040,164.741,61.039,160.714
C06249=1012.931,-102.039,-106.031,164.738,61.044,160.714
C06250=1012.925,-102.333,-106.022,164.736,61.050,160.715
C06251=1012.920,-102.626,-106.013,164.732,61.055,160.714
C06252=1012.915,-102.920,-106.003,164.729,61.061,160.715
C06253=1012.910,-103.170,-105.995,164.728,61.066,160.715
C06254=1012.906,-103.420,-105.988,164.726,61.070,160.715
C06255=1012.902,-103.669,-105.981,164.723,61.074,160.715
C06256=1012.897,-103.919,-105.973,164.721,61.080,160.715
C06257=1012.892,-104.169,-105.965,164.718,61.084,160.715
C06258=1012.888,-104.419,-105.958,164.716,61.088,160.715
C06259=1012.883,-104.669,-105.950,164.714,61.092,160.716
C06260=1012.879,-104.919,-105.943,164.712,61.097,160.716
C06261=1012.874,-105.168,-105.936,164.709,61.102,160.716
C06262=1012.870,-105.419,-105.927,164.707,61.106,160.716
C06263=1012.866,-105.669,-105.920,164.704,61.110,160.716
C06264=1012.861,-105.918,-105.912,164.702,61.114,160.716
C06265=1012.857,-106.168,-105.905,164.700,61.118,160.716
C06266=1012.852,-106.418,-105.897,164.698,61.123,160.716
C06267=1012.848,-106.668,-105.890,164.696,61.127,160.717
C06268=1012.843,-106.918,-105.882,164.693,61.132,160.716
C06269=1012.844,-94.477,-106.693,164.795,61.158,160.755
C06270=1012.847,-94.228,-106.702,164.797,61.153,160.754
C06271=1012.852,-93.977,-106.710,164.799,61.149,160.754
C06272=1012.856,-93.728,-106.718,164.801,61.145,160.754
C06273=1012.861,-93.478,-106.726,164.804,61.139,160.754
C06274=1012.866,-93.229,-106.734,164.806,61.135,160.754
C06275=1012.870,-92.978,-106.743,164.808,61.130,160.754
C06276=1012.875,-92.729,-106.751,164.811,61.126,160.754
C06277=1012.879,-92.478,-106.759,164.813,61.121,160.754
C06278=1012.884,-92.229,-106.767,164.815,61.116,160.753
C06279=1012.889,-91.979,-106.775,164.818,61.112,160.754
C06280=1012.893,-91.730,-106.784,164.820,61.107,160.753
C06281=1012.898,-91.479,-106.791,164.822,61.103,160.753
C06282=1012.901,-91.230,-106.800,164.825,61.097,160.753
C06283=1012.906,-90.980,-106.808,164.826,61.092,160.752
C06284=1012.911,-90.731,-106.816,164.830,61.088,160.753
C06285=1012.915,-90.480,-106.824,164.831,61.083,160.752
C06286=1012.920,-90.231,-106.833,164.835,61.078,160.752
C06287=1012.924,-89.980,-106.841,164.836,61.073,160.752
C06288=1012.929,-89.731,-106.849,164.839,61.068,160.752
C06289=1012.934,-89.481,-106.857,164.841,61.064,160.752
C06290=1012.938,-89.231,-106.866,164.844,61.058,160.751
C06291=1012.943,-88.982,-106.874,164.845,61.053,160.751
C06292=1012.947,-88.731,-106.882,164.849,61.049,160.751
C06293=1012.952,-88.482,-106.890,164.850,61.044,160.751
C06294=1012.957,-88.232,-106.898,164.853,61.038,160.750
C06295=1012.961,-87.982,-106.907,164.854,61.034,160.750
C06296=1012.966,-87.732,-106.915,164.858,61.029,160.750
C06297=1012.970,-87.482,-106.924,164.859,61.024,160.750
C06298=1012.974,-87.256,-106.932,164.861,61.019,160.749
C06299=1012.979,-87.030,-106.938,164.864,61.014,160.750
C06300=1012.983,-86.804,-106.946,164.866,61.010,160.749
C06301=1012.987,-86.578,-106.954,164.868,61.005,160.749
C06302=1012.991,-86.352,-106.962,164.870,61.000,160.749
C06303=1012.995,-86.125,-106.969,164.872,60.996,160.748
C06304=1013.000,-85.899,-106.976,164.874,60.991,160.748
C06305=1013.004,-85.673,-106.984,164.877,60.987,160.748
C06306=1013.008,-85.422,-106.992,164.878,60.982,160.748
C06307=1013.013,-85.173,-107.000,164.881,60.976,160.748
C06308=1013.017,-84.923,-107.009,164.884,60.971,160.747
C06309=1013.022,-84.673,-107.017,164.886,60.966,160.747
C06310=1013.027,-84.424,-107.025,164.888,60.961,160.747
C06311=1013.032,-84.174,-107.034,164.890,60.955,160.747
C06312=1013.037,-83.924,-107.043,164.893,60.950,160.746
C06313=1013.040,-83.674,-107.051,164.895,60.945,160.746
C06314=1013.046,-83.425,-107.059,164.897,60.940,160.746
C06315=1013.051,-83.175,-107.068,164.900,60.934,160.746
C06316=1013.055,-82.924,-107.076,164.903,60.929,160.745
C06317=1013.060,-82.675,-107.084,164.905,60.924,160.745
C06318=1013.064,-82.425,-107.093,164.906,60.918,160.744
C06319=1013.070,-82.175,-107.102,164.909,60.912,160.744
C06320=1013.073,-81.926,-107.110,164.911,60.907,160.744
C06321=1013.079,-81.676,-107.118,164.914,60.902,160.744
C06322=1013.084,-81.426,-107.127,164.917,60.896,160.744
C06323=1013.088,-81.176,-107.136,164.917,60.891,160.743
C06324=1013.093,-80.926,-107.143,164.920,60.885,160.743
C06325=1013.097,-80.676,-107.152,164.923,60.880,160.742
C06326=1013.102,-80.427,-107.161,164.925,60.875,160.742
C06327=1013.107,-80.177,-107.170,164.928,60.869,160.742
C06328=1013.111,-79.927,-107.179,164.930,60.863,160.741
C06329=1013.116,-79.678,-107.187,164.932,60.858,160.741
C06330=1013.121,-79.428,-107.196,164.934,60.853,160.741
C06331=1013.125,-79.178,-107.205,164.937,60.847,160.741
C06332=1013.129,-78.927,-107.214,164.940,60.842,160.740
C06333=1013.134,-78.678,-107.222,164.942,60.837,160.740
C06334=1013.139,-78.428,-107.231,164.944,60.831,160.740
C06335=1013.143,-78.178,-107.240,164.947,60.825,160.739
C06336=1013.148,-77.928,-107.248,164.948,60.820,160.739
C06337=1013.153,-77.678,-107.257,164.951,60.815,160.739
C06338=1013.157,-77.429,-107.266,164.953,60.809,160.738
C06339=1013.162,-77.179,-107.275,164.956,60.803,160.738
C06340=1013.167,-76.929,-107.284,164.958,60.798,160.738
C06341=1013.172,-76.680,-107.294,164.960,60.792,160.737
C06342=1013.176,-76.430,-107.303,164.963,60.787,160.737
C06343=1013.181,-76.180,-107.311,164.965,60.780,160.737
C06344=1013.185,-75.931,-107.320,164.968,60.775,160.736
C06345=1013.190,-75.681,-107.329,164.970,60.770,160.736
C06346=1013.195,-75.431,-107.337,164.972,60.764,160.736
C06347=1013.200,-75.181,-107.346,164.975,60.758,160.735
C06348=1013.204,-74.931,-107.356,164.977,60.752,160.735
C06349=1013.209,-74.681,-107.365,164.980,60.747,160.735
C06350=1013.213,-74.431,-107.374,164.982,60.741,160.734
C06351=1013.217,-74.182,-107.383,164.984,60.735,160.734
C06352=1013.222,-73.932,-107.392,164.987,60.730,160.734
C06353=1013.226,-73.682,-107.401,164.988,60.725,160.733
C06354=1013.231,-73.432,-107.410,164.990,60.719,160.733
C06355=1013.236,-73.183,-107.420,164.993,60.713,160.732
C06356=1013.240,-72.933,-107.429,164.995,60.707,160.732
C06357=1013.245,-72.682,-107.438,164.998,60.702,160.732
C06358=1013.250,-72.433,-107.448,165.000,60.697,160.732
C06359=1013.254,-72.183,-107.457,165.002,60.690,160.731
C06360=1013.259,-71.933,-107.466,165.005,60.685,160.731
C06361=1013.263,-71.684,-107.476,165.007,60.679,160.730
C06362=1013.267,-71.434,-107.485,165.010,60.674,160.730
C06363=1013.272,-71.184,-107.494,165.012,60.668,160.729
C06364=1013.277,-70.935,-107.504,165.014,60.662,160.729
C06365=1013.281,-70.685,-107.513,165.016,60.656,160.729
C06366=1013.287,-70.409,-107.523,165.019,60.649,160.728
C06367=1013.292,-70.133,-107.534,165.022,60.643,160.728
C06368=1013.297,-69.857,-107.543,165.024,60.637,160.728
C06369=1013.302,-69.581,-107.554,165.027,60.630,160.727
C06370=1013.307,-69.331,-107.564,165.029,60.624,160.727
C06371=1013.311,-69.081,-107.573,165.032,60.619,160.726
C06372=1013.316,-68.831,-107.582,165.034,60.613,160.726
C06373=1013.320,-68.582,-107.592,165.036,60.607,160.725
C06374=1013.325,-68.332,-107.601,165.038,60.600,160.725
C06375=1013.330,-68.083,-107.611,165.042,60.595,160.725
C06376=1013.334,-67.833,-107.620,165.044,60.588,160.724
C06377=1013.339,-67.583,-107.629,165.046,60.582,160.724
C06378=1013.344,-67.333,-107.638,165.048,60.577,160.724
C06379=1013.348,-67.083,-107.648,165.050,60.571,160.723
C06380=1013.353,-66.834,-107.657,165.052,60.565,160.722
C06381=1013.358,-66.584,-107.666,165.055,60.558,160.722
C06382=1013.362,-66.334,-107.676,165.057,60.552,160.722
C06383=1013.367,-66.084,-107.685,165.060,60.547,160.721
C06384=1013.372,-65.835,-107.695,165.062,60.541,160.721
C06385=1013.376,-65.585,-107.704,165.065,60.534,160.720
C06386=1013.381,-65.335,-107.714,165.067,60.528,160.720
C06387=1013.386,-65.085,-107.723,165.069,60.522,160.719
C06388=1013.390,-64.836,-107.733,165.071,60.516,160.719
C06389=1013.395,-64.586,-107.742,165.074,60.509,160.718
C06390=1013.400,-64.337,-107.752,165.076,60.503,160.718
C06391=1013.404,-64.087,-107.761,165.078,60.497,160.717
C06392=1013.409,-63.837,-107.771,165.081,60.491,160.717
C06393=1013.414,-63.586,-107.780,165.083,60.484,160.716
C06394=1013.419,-63.337,-107.790,165.085,60.478,160.716
C06395=1013.424,-63.087,-107.799,165.088,60.472,160.716
C06396=1013.428,-62.838,-107.809,165.090,60.466,160.715
C06397=1013.433,-62.587,-107.818,165.092,60.460,160.714
C06398=1013.438,-62.338,-107.828,165.095,60.453,160.714
C06399=1013.442,-62.088,-107.837,165.097,60.447,160.714
C06400=1013.447,-61.839,-107.846,165.100,60.440,160.713
C06401=1013.452,-61.589,-107.856,165.102,60.434,160.713
C06402=1013.457,-61.339,-107.866,165.104,60.428,160.712
C06403=1013.462,-61.089,-107.876,165.108,60.422,160.712
C06404=1013.467,-60.839,-107.885,165.109,60.415,160.711
C06405=1013.471,-60.590,-107.894,165.112,60.408,160.711
C06406=1013.476,-60.340,-107.904,165.114,60.402,160.710
C06407=1013.481,-60.090,-107.913,165.117,60.396,160.710
C06408=1013.485,-59.841,-107.924,165.119,60.390,160.709
C06409=1013.490,-59.590,-107.933,165.121,60.382,160.708
C06410=1013.495,-59.340,-107.943,165.123,60.376,160.708
C06411=1013.500,-59.091,-107.953,165.127,60.370,160.708
C06412=1013.504,-58.841,-107.962,165.129,60.363,160.707
C06413=1013.509,-58.592,-107.972,165.131,60.356,160.706
C06414=1013.514,-58.342,-107.981,165.133,60.350,160.706
C06415=1013.519,-58.091,-107.991,165.136,60.344,160.706
C06416=1013.524,-57.842,-108.001,165.137,60.337,160.705
C06417=1013.529,-57.593,-108.010,165.140,60.330,160.704
C06418=1013.533,-57.343,-108.019,165.142,60.324,160.704
C06419=1013.538,-57.093,-108.029,165.145,60.317,160.703
C06420=1013.543,-56.843,-108.039,165.147,60.311,160.702
C06421=1013.548,-56.593,-108.049,165.149,60.303,160.702
C06422=1013.553,-56.344,-108.058,165.152,60.297,160.701
C06423=1013.558,-56.094,-108.068,165.154,60.291,160.701
C06424=1013.563,-55.844,-108.078,165.157,60.283,160.700
C06425=1013.568,-55.594,-108.087,165.160,60.277,160.700
C06426=1013.572,-55.345,-108.097,165.161,60.270,160.699
C06427=1013.577,-55.095,-108.107,165.164,60.264,160.699
C06428=1013.583,-54.845,-108.117,165.166,60.257,160.698
C06429=1013.587,-54.595,-108.126,165.169,60.250,160.697
C06430=1013.592,-54.320,-108.138,165.171,60.242,160.696
C06431=1013.597,-54.046,-108.148,165.174,60.234,160.696
C06432=1013.603,-53.771,-108.159,165.176,60.227,160.695
C06433=1013.609,-53.496,-108.170,165.179,60.220,160.695
C06434=1013.613,-53.247,-108.179,165.181,60.213,160.694
C06435=1013.619,-52.996,-108.189,165.184,60.206,160.694
C06436=1013.623,-52.747,-108.199,165.186,60.199,160.693
C06437=1013.628,-52.497,-108.208,165.188,60.192,160.692
C06438=1013.633,-52.248,-108.218,165.191,60.185,160.692
C06439=1013.638,-51.998,-108.228,165.194,60.178,160.691
C06440=1013.643,-51.748,-108.237,165.195,60.171,160.690
C06441=1013.648,-51.498,-108.247,165.198,60.165,160.690
C06442=1013.653,-51.248,-108.258,165.201,60.158,160.689
C06443=1013.657,-50.998,-108.268,165.203,60.150,160.689
C06444=1013.662,-50.748,-108.279,165.205,60.144,160.688
C06445=1013.667,-50.498,-108.288,165.208,60.137,160.687
C06446=1013.671,-50.249,-108.299,165.210,60.131,160.687
C06447=1013.676,-49.999,-108.309,165.212,60.124,160.686
C06448=1013.681,-49.749,-108.319,165.215,60.117,160.686
C06449=1013.686,-49.499,-108.329,165.216,60.110,160.685
C06450=1013.691,-49.250,-108.340,165.219,60.103,160.684
C06451=1013.695,-49.000,-108.350,165.222,60.096,160.684
C06452=1013.701,-48.750,-108.361,165.223,60.090,160.683
C06453=1013.705,-48.501,-108.371,165.227,60.083,160.683
C06454=1013.710,-48.251,-108.381,165.229,60.076,160.682
C06455=1013.714,-48.001,-108.391,165.231,60.069,160.681
C06456=1013.719,-47.751,-108.401,165.233,60.062,160.681
C06457=1013.724,-47.501,-108.412,165.236,60.055,160.680
C06458=1013.729,-47.252,-108.423,165.238,60.048,160.679
C06459=1013.734,-47.003,-108.432,165.241,60.041,160.679
C06460=1013.738,-46.752,-108.443,165.243,60.035,160.678
C06461=1013.743,-46.503,-108.453,165.245,60.027,160.678
C06462=1013.748,-46.252,-108.464,165.248,60.020,160.677
C06463=1013.753,-46.004,-108.474,165.250,60.013,160.676
C06464=1013.758,-45.753,-108.485,165.252,60.007,160.676
C06465=1013.763,-45.504,-108.495,165.255,60.000,160.675
C06466=1013.767,-45.254,-108.505,165.257,59.992,160.674
C06467=1013.772,-45.004,-108.515,165.260,59.985,160.674
C06468=1013.777,-44.755,-108.526,165.262,59.978,160.673
C06469=1013.782,-44.505,-108.537,165.263,59.971,160.672
C06470=1013.786,-44.255,-108.547,165.267,59.964,160.672
C06471=1013.791,-44.005,-108.557,165.269,59.957,160.671
C06472=1013.796,-43.756,-108.568,165.272,59.950,160.670
C06473=1013.801,-43.506,-108.578,165.274,59.943,160.670
C06474=1013.806,-43.256,-108.588,165.276,59.935,160.669
///RCONF 1,0,0,0,0,0,0,0,0,0,0,0,0,0,0,0,0,0,0,0,0,0,0,0
C06475=1013.811,-43.006,-108.599,165.279,59.928,160.668
C06476=1013.816,-42.757,-108.609,165.280,59.921,160.667
C06477=1013.821,-42.507,-108.620,165.283,59.914,160.667
C06478=1013.826,-42.257,-108.630,165.285,59.907,160.666
C06479=1013.830,-42.007,-108.641,165.288,59.900,160.665
C06480=1013.835,-41.758,-108.651,165.290,59.892,160.665
C06481=1013.840,-41.508,-108.662,165.293,59.885,160.664
C06482=1013.845,-41.258,-108.672,165.295,59.878,160.663
C06483=1013.850,-41.008,-108.683,165.298,59.871,160.663
C06484=1013.855,-40.759,-108.693,165.300,59.863,160.662
C06485=1013.859,-40.509,-108.704,165.303,59.856,160.661
C06486=1013.865,-40.260,-108.714,165.304,59.848,160.660
C06487=1013.869,-40.009,-108.725,165.307,59.841,160.660
C06488=1013.874,-39.760,-108.735,165.309,59.834,160.659
C06489=1013.879,-39.510,-108.746,165.312,59.826,160.658
C06490=1013.884,-39.260,-108.756,165.314,59.819,160.658
C06491=1013.889,-39.011,-108.768,165.317,59.812,160.657
C06492=1013.894,-38.761,-108.778,165.318,59.805,160.656
C06493=1013.898,-38.511,-108.789,165.321,59.798,160.656
C06494=1013.903,-38.237,-108.802,165.324,59.789,160.655
C06495=1013.909,-37.962,-108.812,165.326,59.782,160.654
C06496=1013.914,-37.687,-108.824,165.329,59.774,160.653
C06497=1013.919,-37.413,-108.837,165.331,59.766,160.652
C06498=1013.924,-37.163,-108.848,165.333,59.759,160.652
C06499=1013.929,-36.913,-108.858,165.336,59.751,160.651
C06500=1013.934,-36.664,-108.869,165.338,59.744,160.650
C06501=1013.939,-36.414,-108.880,165.341,59.737,160.650
C06502=1013.943,-36.164,-108.891,165.343,59.730,160.649
C06503=1013.948,-35.915,-108.903,165.346,59.722,160.648
C06504=1013.953,-35.665,-108.912,165.348,59.714,160.647
C06505=1013.958,-35.415,-108.924,165.350,59.707,160.647
C06506=1013.963,-35.165,-108.935,165.353,59.700,160.646
C06507=1013.967,-34.916,-108.946,165.355,59.693,160.645
C06508=1013.973,-34.666,-108.957,165.358,59.686,160.645
C06509=1013.978,-34.416,-108.967,165.359,59.678,160.644
C06510=1013.982,-34.167,-108.978,165.362,59.670,160.643
C06511=1013.987,-33.916,-108.989,165.364,59.663,160.642
C06512=1013.993,-33.667,-109.000,165.366,59.655,160.641
C06513=1013.997,-33.418,-109.011,165.369,59.648,160.641
C06514=1014.002,-33.167,-109.022,165.371,59.641,160.640
C06515=1014.007,-32.918,-109.033,165.374,59.632,160.639
C06516=1014.012,-32.669,-109.044,165.377,59.625,160.639
C06517=1014.017,-32.418,-109.055,165.379,59.618,160.638
C06518=1014.022,-32.169,-109.066,165.381,59.610,160.637
C06519=1014.026,-31.920,-109.077,165.384,59.603,160.636
C06520=1014.031,-31.669,-109.088,165.386,59.595,160.636
C06521=1014.036,-31.420,-109.099,165.388,59.587,160.635
C06522=1014.041,-31.170,-109.110,165.391,59.580,160.634
C06523=1014.046,-30.921,-109.122,165.392,59.572,160.633
C06524=1014.050,-30.670,-109.132,165.396,59.565,160.632
C06525=1014.056,-30.421,-109.143,165.398,59.557,160.631
C06526=1014.061,-30.172,-109.154,165.400,59.549,160.631
C06527=1014.065,-29.921,-109.165,165.402,59.542,160.630
C06528=1014.070,-29.671,-109.176,165.405,59.534,160.629
C06529=1014.076,-29.422,-109.187,165.407,59.526,160.628
C06530=1014.080,-29.173,-109.198,165.410,59.519,160.628
C06531=1014.085,-28.922,-109.209,165.412,59.511,160.627
C06532=1014.090,-28.673,-109.221,165.415,59.504,160.626
C06533=1014.096,-28.423,-109.232,165.417,59.496,160.625
C06534=1014.100,-28.174,-109.243,165.418,59.488,160.624
C06535=1014.105,-27.924,-109.253,165.422,59.480,160.624
C06536=1014.110,-27.674,-109.265,165.424,59.472,160.623
C06537=1014.115,-27.424,-109.276,165.426,59.465,160.622
C06538=1014.120,-27.174,-109.288,165.428,59.457,160.621
C06539=1014.125,-26.924,-109.299,165.431,59.450,160.620
C06540=1014.129,-26.675,-109.310,165.433,59.442,160.620
C06541=1014.134,-26.426,-109.322,165.435,59.435,160.619
C06542=1014.139,-26.176,-109.333,165.438,59.427,160.618
C06543=1014.144,-25.926,-109.345,165.441,59.419,160.617
C06544=1014.149,-25.676,-109.356,165.443,59.411,160.616
C06545=1014.154,-25.427,-109.367,165.445,59.404,160.616
C06546=1014.159,-25.177,-109.379,165.447,59.396,160.615
C06547=1014.163,-24.927,-109.391,165.450,59.389,160.614
C06548=1014.168,-24.677,-109.402,165.452,59.381,160.613
C06549=1014.173,-24.428,-109.414,165.455,59.373,160.612
C06550=1014.178,-24.178,-109.425,165.457,59.365,160.611
C06551=1014.182,-23.929,-109.436,165.459,59.357,160.610
C06552=1014.187,-23.679,-109.448,165.462,59.350,160.610
C06553=1014.192,-23.429,-109.459,165.463,59.342,160.609
C06554=1014.197,-23.179,-109.471,165.466,59.334,160.608
C06555=1014.202,-22.929,-109.482,165.469,59.327,160.607
C06556=1014.207,-22.680,-109.494,165.471,59.319,160.606
C06557=1014.212,-22.430,-109.505,165.473,59.311,160.605
C06558=1014.218,-22.154,-109.518,165.476,59.302,160.605
C06559=1014.223,-21.879,-109.531,165.478,59.293,160.604
C06560=1014.229,-21.603,-109.544,165.481,59.285,160.603
C06561=1014.234,-21.328,-109.556,165.484,59.276,160.602
C06562=1014.239,-21.078,-109.568,165.486,59.268,160.601
C06563=1014.244,-20.828,-109.580,165.489,59.260,160.600
C06564=1014.249,-20.578,-109.591,165.491,59.252,160.599
C06565=1014.254,-20.329,-109.603,165.493,59.244,160.598
C06566=1014.258,-20.080,-109.614,165.497,59.237,160.598
C06567=1014.263,-19.830,-109.625,165.498,59.229,160.597
C06568=1014.268,-19.580,-109.637,165.500,59.221,160.596
C06569=1014.273,-19.331,-109.649,165.503,59.212,160.595
C06570=1014.278,-19.081,-109.661,165.505,59.204,160.594
C06571=1014.283,-18.831,-109.672,165.507,59.197,160.593
C06572=1014.288,-18.581,-109.684,165.510,59.188,160.592
C06573=1014.293,-18.332,-109.695,165.512,59.180,160.591
C06574=1014.298,-18.082,-109.706,165.514,59.172,160.590
C06575=1014.304,-17.833,-109.719,165.517,59.164,160.590
C06576=1014.309,-17.583,-109.730,165.520,59.157,160.589
C06577=1014.314,-17.333,-109.742,165.522,59.149,160.588
C06578=1014.319,-17.083,-109.753,165.525,59.141,160.587
C06579=1014.324,-16.833,-109.765,165.527,59.133,160.586
C06580=1014.328,-16.584,-109.777,165.530,59.124,160.585
C06581=1014.333,-16.334,-109.789,165.532,59.116,160.584
C06582=1014.338,-16.084,-109.800,165.533,59.108,160.583
C06583=1014.343,-15.834,-109.812,165.537,59.100,160.583
C06584=1014.348,-15.585,-109.825,165.538,59.092,160.582
C06585=1014.353,-15.335,-109.836,165.540,59.084,160.581
C06586=1014.358,-15.085,-109.847,165.543,59.076,160.580
C06587=1014.362,-14.836,-109.860,165.545,59.068,160.579
C06588=1014.367,-14.586,-109.872,165.547,59.060,160.578
C06589=1014.373,-14.337,-109.884,165.550,59.052,160.577
C06590=1014.377,-14.087,-109.896,165.552,59.044,160.576
C06591=1014.382,-13.837,-109.907,165.554,59.036,160.575
C06592=1014.387,-13.588,-109.920,165.558,59.028,160.575
C06593=1014.392,-13.338,-109.932,165.560,59.021,160.574
C06594=1014.397,-13.088,-109.944,165.562,59.013,160.573
C06595=1014.402,-12.839,-109.955,165.565,59.004,160.572
C06596=1014.406,-12.589,-109.968,165.567,58.996,160.571
C06597=1014.411,-12.339,-109.980,165.570,58.988,160.570
C06598=1014.416,-12.090,-109.991,165.571,58.979,160.569
C06599=1014.421,-11.840,-110.004,165.573,58.972,160.568
C06600=1014.427,-11.590,-110.016,165.576,58.963,160.567
C06601=1014.432,-11.340,-110.028,165.578,58.955,160.566
C06602=1014.436,-11.090,-110.040,165.581,58.947,160.566
C06603=1014.441,-10.841,-110.052,165.583,58.939,160.565
C06604=1014.446,-10.591,-110.064,165.585,58.931,160.564
C06605=1014.451,-10.342,-110.076,165.588,58.923,160.563
C06606=1014.456,-10.092,-110.088,165.590,58.915,160.562
C06607=1014.461,-9.843,-110.101,165.593,58.907,160.561
C06608=1014.466,-9.593,-110.112,165.595,58.898,160.560
C06609=1014.471,-9.344,-110.124,165.598,58.890,160.559
C06610=1014.475,-9.093,-110.136,165.600,58.882,160.558
C06611=1014.481,-8.844,-110.149,165.603,58.874,160.557
C06612=1014.486,-8.594,-110.161,165.605,58.866,160.556
C06613=1014.491,-8.344,-110.173,165.607,58.857,160.555
C06614=1014.496,-8.095,-110.185,165.609,58.849,160.554
C06615=1014.501,-7.845,-110.197,165.611,58.841,160.553
C06616=1014.506,-7.596,-110.210,165.614,58.833,160.553
C06617=1014.511,-7.346,-110.221,165.617,58.823,160.551
C06618=1014.516,-7.097,-110.233,165.619,58.816,160.550
C06619=1014.521,-6.847,-110.246,165.622,58.807,160.550
C06620=1014.526,-6.597,-110.258,165.623,58.799,160.548
C06621=1014.531,-6.348,-110.270,165.626,58.790,160.548
C06622=1014.537,-6.070,-110.284,165.629,58.781,160.547
C06623=1014.541,-5.792,-110.297,165.631,58.772,160.545
C06624=1014.548,-5.515,-110.311,165.634,58.763,160.544
C06625=1014.553,-5.237,-110.325,165.636,58.753,160.543
C06626=1014.558,-4.988,-110.337,165.638,58.745,160.542
C06627=1014.563,-4.739,-110.348,165.642,58.737,160.541
C06628=1014.568,-4.488,-110.361,165.643,58.728,160.540
C06629=1014.573,-4.239,-110.374,165.646,58.720,160.539
C06630=1014.578,-3.989,-110.386,165.648,58.712,160.538
C06631=1014.582,-3.740,-110.398,165.651,58.704,160.538
C06632=1014.588,-3.489,-110.412,165.653,58.696,160.537
C06633=1014.593,-3.240,-110.424,165.655,58.687,160.535
C06634=1014.597,-2.991,-110.437,165.658,58.679,160.535
C06635=1014.602,-2.741,-110.449,165.660,58.671,160.534
C06636=1014.607,-2.492,-110.462,165.663,58.663,160.533
C06637=1014.613,-2.242,-110.475,165.664,58.654,160.532
C06638=1014.617,-1.992,-110.487,165.667,58.646,160.531
C06639=1014.621,-1.742,-110.499,165.669,58.638,160.530
C06640=1014.626,-1.493,-110.512,165.672,58.630,160.529
C06641=1014.632,-1.243,-110.525,165.674,58.621,160.528
C06642=1014.636,-0.993,-110.538,165.677,58.613,160.527
C06643=1014.641,-0.744,-110.550,165.679,58.605,160.526
C06644=1014.646,-0.495,-110.563,165.681,58.596,160.525
C06645=1014.651,-0.244,-110.576,165.684,58.588,160.524
C06646=1014.656,0.005,-110.589,165.687,58.580,160.523
C06647=1014.661,0.255,-110.601,165.688,58.571,160.522
C06648=1014.666,0.504,-110.613,165.691,58.563,160.521
C06649=1014.671,0.754,-110.627,165.693,58.554,160.520
C06650=1014.676,1.003,-110.639,165.696,58.546,160.519
C06651=1014.680,1.253,-110.652,165.698,58.538,160.518
C06652=1014.686,1.503,-110.665,165.700,58.529,160.517
C06653=1014.691,1.752,-110.678,165.702,58.521,160.516
C06654=1014.695,2.002,-110.690,165.705,58.512,160.515
C06655=1014.700,2.251,-110.703,165.707,58.505,160.514
C06656=1014.706,2.501,-110.716,165.709,58.496,160.513
C06657=1014.710,2.751,-110.728,165.711,58.488,160.512
C06658=1014.715,3.000,-110.741,165.714,58.479,160.511
C06659=1014.721,3.250,-110.754,165.717,58.470,160.510
C06660=1014.725,3.500,-110.767,165.719,58.462,160.509
C06661=1014.730,3.749,-110.779,165.722,58.454,160.508
C06662=1014.735,3.999,-110.792,165.723,58.445,160.507
C06663=1014.740,4.248,-110.805,165.726,58.437,160.506
C06664=1014.745,4.498,-110.817,165.729,58.428,160.505
C06665=1014.750,4.748,-110.831,165.731,58.420,160.504
C06666=1014.755,4.998,-110.843,165.733,58.411,160.503
C06667=1014.760,5.247,-110.856,165.735,58.402,160.502
C06668=1014.765,5.497,-110.869,165.738,58.394,160.501
C06669=1014.770,5.746,-110.882,165.740,58.385,160.500
C06670=1014.774,5.996,-110.894,165.743,58.377,160.499
C06671=1014.780,6.246,-110.907,165.745,58.368,160.498
C06672=1014.785,6.495,-110.920,165.748,58.359,160.497
C06673=1014.790,6.746,-110.933,165.750,58.351,160.496
C06674=1014.795,6.995,-110.946,165.752,58.342,160.495
C06675=1014.800,7.244,-110.958,165.755,58.333,160.494
C06676=1014.805,7.494,-110.972,165.757,58.326,160.493
C06677=1014.810,7.743,-110.984,165.759,58.317,160.492
C06678=1014.815,7.993,-110.998,165.762,58.308,160.491
C06679=1014.820,8.243,-111.010,165.763,58.299,160.490
C06680=1014.825,8.492,-111.023,165.767,58.291,160.489
C06681=1014.830,8.742,-111.036,165.769,58.282,160.488
C06682=1014.835,8.992,-111.048,165.771,58.273,160.487
C06683=1014.841,9.241,-111.062,165.773,58.264,160.486
C06684=1014.845,9.491,-111.074,165.776,58.255,160.484
C06685=1014.850,9.740,-111.087,165.779,58.247,160.484
C06686=1014.856,10.019,-111.102,165.781,58.237,160.482
C06687=1014.862,10.300,-111.116,165.784,58.227,160.481
C06688=1014.868,10.579,-111.131,165.786,58.218,160.480
C06689=1014.873,10.858,-111.146,165.790,58.208,160.479
C06690=1014.879,11.108,-111.158,165.792,58.199,160.478
C06691=1014.883,11.358,-111.171,165.794,58.191,160.477
C06692=1014.888,11.608,-111.184,165.796,58.182,160.476
C06693=1014.893,11.857,-111.197,165.799,58.173,160.474
C06694=1014.899,12.107,-111.210,165.801,58.164,160.473
C06695=1014.904,12.356,-111.223,165.803,58.155,160.472
C06696=1014.909,12.606,-111.236,165.805,58.146,160.471
C06697=1014.913,12.856,-111.249,165.808,58.137,160.470
C06698=1014.920,13.105,-111.262,165.811,58.128,160.469
C06699=1014.924,13.355,-111.276,165.813,58.121,160.468
C06700=1014.929,13.605,-111.289,165.815,58.112,160.467
C06701=1014.934,13.854,-111.302,165.818,58.103,160.466
C06702=1014.939,14.104,-111.315,165.819,58.094,160.465
C06703=1014.943,14.354,-111.328,165.823,58.086,160.464
C06704=1014.949,14.603,-111.342,165.825,58.077,160.463
C06705=1014.953,14.853,-111.355,165.827,58.068,160.462
C06706=1014.959,15.102,-111.369,165.829,58.059,160.461
C06707=1014.963,15.352,-111.381,165.832,58.050,160.460
C06708=1014.969,15.601,-111.395,165.833,58.042,160.458
C06709=1014.973,15.851,-111.408,165.837,58.034,160.458
C06710=1014.979,16.100,-111.422,165.839,58.025,160.456
C06711=1014.983,16.350,-111.435,165.842,58.016,160.455
C06712=1014.989,16.600,-111.448,165.843,58.007,160.454
C06713=1014.994,16.850,-111.462,165.846,57.998,160.453
C06714=1014.999,17.099,-111.474,165.849,57.989,160.452
C06715=1015.004,17.349,-111.488,165.851,57.980,160.451
C06716=1015.009,17.598,-111.501,165.853,57.972,160.450
C06717=1015.014,17.848,-111.515,165.855,57.963,160.449
C06718=1015.019,18.097,-111.528,165.858,57.954,160.448
C06719=1015.024,18.347,-111.542,165.861,57.945,160.447
C06720=1015.029,18.596,-111.554,165.862,57.937,160.445
C06721=1015.034,18.846,-111.569,165.865,57.928,160.444
C06722=1015.039,19.096,-111.583,165.868,57.920,160.444
C06723=1015.044,19.345,-111.596,165.870,57.911,160.442
C06724=1015.049,19.595,-111.609,165.872,57.902,160.441
C06725=1015.054,19.844,-111.622,165.875,57.893,160.440
C06726=1015.058,20.094,-111.637,165.878,57.884,160.439
C06727=1015.064,20.344,-111.650,165.879,57.876,160.438
C06728=1015.068,20.593,-111.663,165.882,57.867,160.437
C06729=1015.074,20.843,-111.677,165.884,57.858,160.436
C06730=1015.079,21.092,-111.691,165.887,57.849,160.435
C06731=1015.083,21.342,-111.704,165.889,57.840,160.434
C06732=1015.089,21.592,-111.718,165.891,57.832,160.433
C06733=1015.094,21.841,-111.732,165.894,57.823,160.431
C06734=1015.099,22.091,-111.745,165.897,57.814,160.430
C06735=1015.104,22.340,-111.758,165.898,57.805,160.429
C06736=1015.108,22.590,-111.773,165.901,57.796,160.428
C06737=1015.114,22.840,-111.786,165.903,57.787,160.427
C06738=1015.118,23.089,-111.799,165.906,57.778,160.426
C06739=1015.124,23.338,-111.813,165.908,57.770,160.425
C06740=1015.129,23.589,-111.827,165.910,57.761,160.424
C06741=1015.133,23.838,-111.841,165.913,57.752,160.423
C06742=1015.139,24.087,-111.854,165.916,57.743,160.422
C06743=1015.144,24.337,-111.868,165.918,57.734,160.420
C06744=1015.149,24.586,-111.881,165.919,57.725,160.419
C06745=1015.154,24.836,-111.895,165.922,57.716,160.418
C06746=1015.159,25.086,-111.909,165.925,57.707,160.417
C06747=1015.164,25.335,-111.923,165.927,57.698,160.416
C06748=1015.169,25.585,-111.936,165.930,57.689,160.415
C06749=1015.174,25.835,-111.950,165.932,57.681,160.414
C06750=1015.180,26.115,-111.966,165.935,57.671,160.413
C06751=1015.185,26.397,-111.981,165.937,57.660,160.411
C06752=1015.191,26.677,-111.997,165.939,57.650,160.410
C06753=1015.196,26.959,-112.012,165.943,57.640,160.409
C06754=1015.202,27.208,-112.026,165.945,57.632,160.408
C06755=1015.207,27.458,-112.040,165.948,57.623,160.407
C06756=1015.212,27.708,-112.055,165.950,57.614,160.405
C06757=1015.216,27.957,-112.067,165.952,57.605,160.404
C06758=1015.221,28.207,-112.082,165.955,57.596,160.403
C06759=1015.227,28.457,-112.096,165.957,57.587,160.402
C06760=1015.231,28.707,-112.110,165.959,57.578,160.401
C06761=1015.236,28.955,-112.124,165.961,57.569,160.400
C06762=1015.241,29.205,-112.138,165.964,57.561,160.399
C06763=1015.246,29.455,-112.152,165.967,57.552,160.398
C06764=1015.251,29.704,-112.165,165.970,57.543,160.397
C06765=1015.256,29.954,-112.180,165.971,57.534,160.395
C06766=1015.262,30.203,-112.194,165.973,57.525,160.394
C06767=1015.266,30.453,-112.208,165.976,57.516,160.393
C06768=1015.271,30.702,-112.222,165.979,57.507,160.392
C06769=1015.276,30.952,-112.236,165.982,57.498,160.391
C06770=1015.281,31.201,-112.250,165.983,57.490,160.390
C06771=1015.286,31.451,-112.265,165.986,57.481,160.389
C06772=1015.292,31.701,-112.278,165.988,57.471,160.387
C06773=1015.296,31.950,-112.292,165.991,57.462,160.386
C06774=1015.301,32.200,-112.306,165.993,57.453,160.385
C06775=1015.306,32.450,-112.321,165.995,57.445,160.384
C06776=1015.311,32.699,-112.335,165.997,57.435,160.383
C06777=1015.317,32.949,-112.349,166.000,57.426,160.382
C06778=1015.321,33.198,-112.363,166.003,57.418,160.381
C06779=1015.327,33.447,-112.376,166.005,57.408,160.379
C06780=1015.331,33.697,-112.391,166.008,57.399,160.378
C06781=1015.337,33.947,-112.405,166.010,57.390,160.377
C06782=1015.342,34.196,-112.420,166.012,57.382,160.376
C06783=1015.347,34.445,-112.433,166.014,57.372,160.375
C06784=1015.351,34.695,-112.448,166.017,57.363,160.374
C06785=1015.357,34.945,-112.462,166.020,57.355,160.373
C06786=1015.362,35.194,-112.476,166.022,57.345,160.371
C06787=1015.367,35.444,-112.490,166.025,57.336,160.370
C06788=1015.372,35.694,-112.505,166.027,57.327,160.369
C06789=1015.377,35.943,-112.518,166.030,57.318,160.368
C06790=1015.381,36.193,-112.533,166.032,57.309,160.367
C06791=1015.387,36.442,-112.546,166.033,57.300,160.366
C06792=1015.392,36.691,-112.562,166.036,57.291,160.364
C06793=1015.397,36.941,-112.576,166.039,57.282,160.363
C06794=1015.402,37.191,-112.590,166.042,57.273,160.362
C06795=1015.407,37.441,-112.604,166.044,57.264,160.361
C06796=1015.411,37.689,-112.619,166.046,57.255,160.360
C06797=1015.417,37.939,-112.633,166.048,57.246,160.359
C06798=1015.422,38.189,-112.647,166.051,57.237,160.358
C06799=1015.427,38.438,-112.663,166.053,57.228,160.357
C06800=1015.431,38.688,-112.677,166.056,57.219,160.356
C06801=1015.437,38.938,-112.691,166.058,57.211,160.354
C06802=1015.442,39.187,-112.705,166.060,57.201,160.353
C06803=1015.447,39.437,-112.721,166.063,57.192,160.352
C06804=1015.452,39.686,-112.734,166.066,57.183,160.351
C06805=1015.456,39.935,-112.749,166.068,57.174,160.350
C06806=1015.461,40.185,-112.764,166.071,57.165,160.349
C06807=1015.466,40.435,-112.778,166.073,57.156,160.348
C06808=1015.471,40.684,-112.792,166.075,57.147,160.346
C06809=1015.477,40.933,-112.807,166.077,57.138,160.345
C06810=1015.484,41.306,-112.829,166.081,57.124,160.343
C06811=1015.492,41.680,-112.850,166.085,57.111,160.342
C06812=1015.499,42.053,-112.873,166.088,57.097,160.340
C06813=1015.506,42.426,-112.894,166.092,57.084,160.338
C06814=1015.512,42.741,-112.913,166.095,57.072,160.337
C06815=1015.518,43.057,-112.932,166.098,57.062,160.335
C06816=1015.523,43.307,-112.947,166.101,57.053,160.334
C06817=1015.528,43.556,-112.962,166.103,57.043,160.333
C06818=1015.533,43.806,-112.976,166.106,57.034,160.332
C06819=1015.538,44.055,-112.992,166.107,57.026,160.331
C06820=1015.543,44.304,-113.007,166.110,57.017,160.330
C06821=1015.547,44.554,-113.021,166.112,57.008,160.328
C06822=1015.553,44.803,-113.036,166.115,56.999,160.327
C06823=1015.557,45.053,-113.051,166.118,56.990,160.326
C06824=1015.562,45.303,-113.066,166.119,56.981,160.325
C06825=1015.567,45.552,-113.080,166.122,56.972,160.324
C06826=1015.572,45.802,-113.096,166.125,56.963,160.323
C06827=1015.577,46.051,-113.111,166.127,56.954,160.322
C06828=1015.582,46.301,-113.125,166.130,56.945,160.321
C06829=1015.587,46.550,-113.140,166.131,56.936,160.319
C06830=1015.592,46.799,-113.156,166.134,56.927,160.318
C06831=1015.597,47.049,-113.170,166.137,56.918,160.317
C06832=1015.602,47.299,-113.185,166.139,56.909,160.316
C06833=1015.606,47.548,-113.200,166.142,56.900,160.315
C06834=1015.612,47.798,-113.215,166.144,56.891,160.314
C06835=1015.617,48.047,-113.230,166.146,56.882,160.312
C06836=1015.621,48.297,-113.245,166.149,56.873,160.311
C06837=1015.626,48.546,-113.260,166.151,56.864,160.310
C06838=1015.631,48.795,-113.275,166.154,56.855,160.309
C06839=1015.636,49.045,-113.289,166.156,56.846,160.308
C06840=1015.641,49.295,-113.305,166.159,56.837,160.307
C06841=1015.646,49.544,-113.320,166.162,56.827,160.305
C06842=1015.651,49.794,-113.334,166.163,56.819,160.304
C06843=1015.656,50.043,-113.349,166.166,56.809,160.303
C06844=1015.661,50.292,-113.364,166.168,56.801,160.302
C06845=1015.666,50.541,-113.380,166.171,56.791,160.301
C06846=1015.671,50.791,-113.394,166.174,56.782,160.300
C06847=1015.676,51.041,-113.409,166.176,56.773,160.298
C06848=1015.681,51.290,-113.424,166.179,56.764,160.297
C06849=1015.686,51.540,-113.439,166.181,56.755,160.296
C06850=1015.691,51.789,-113.454,166.184,56.746,160.295
C06851=1015.696,52.038,-113.469,166.185,56.737,160.294
C06852=1015.701,52.288,-113.485,166.188,56.727,160.292
C06853=1015.706,52.538,-113.499,166.190,56.718,160.291
C06854=1015.711,52.787,-113.514,166.193,56.709,160.290
C06855=1015.716,53.037,-113.530,166.196,56.700,160.289
C06856=1015.721,53.286,-113.545,166.198,56.691,160.288
C06857=1015.726,53.536,-113.559,166.200,56.681,160.286
C06858=1015.731,53.785,-113.574,166.203,56.672,160.285
C06859=1015.736,54.034,-113.590,166.205,56.663,160.284
C06860=1015.740,54.284,-113.605,166.208,56.653,160.283
C06861=1015.746,54.534,-113.621,166.211,56.645,160.282
C06862=1015.751,54.784,-113.635,166.213,56.635,160.281
C06863=1015.756,55.033,-113.651,166.216,56.626,160.280
C06864=1015.761,55.282,-113.666,166.218,56.617,160.278
C06865=1015.766,55.532,-113.681,166.221,56.608,160.277
C06866=1015.771,55.781,-113.696,166.223,56.598,160.276
C06867=1015.776,56.031,-113.711,166.226,56.589,160.275
C06868=1015.781,56.280,-113.726,166.228,56.580,160.273
C06869=1015.786,56.530,-113.741,166.231,56.570,160.272
C06870=1015.791,56.779,-113.756,166.233,56.562,160.271
C06871=1015.796,57.029,-113.772,166.236,56.552,160.270
C06872=1015.802,57.278,-113.787,166.238,56.543,160.269
C06873=1015.806,57.528,-113.801,166.241,56.533,160.267
C06874=1015.811,57.777,-113.816,166.243,56.524,160.266
C06875=1015.817,58.027,-113.832,166.246,56.515,160.265
C06876=1015.822,58.307,-113.849,166.248,56.505,160.263
C06877=1015.828,58.589,-113.866,166.251,56.494,160.262
C06878=1015.834,58.870,-113.883,166.253,56.484,160.261
C06879=1015.839,59.152,-113.900,166.256,56.473,160.259
C06880=1015.845,59.401,-113.915,166.259,56.464,160.258
C06881=1015.850,59.650,-113.930,166.262,56.455,160.257
C06882=1015.855,59.900,-113.946,166.264,56.445,160.256
C06883=1015.860,60.149,-113.961,166.266,56.436,160.255
C06884=1015.865,60.399,-113.976,166.269,56.426,160.253
C06885=1015.870,60.648,-113.992,166.271,56.417,160.252
C06886=1015.875,60.897,-114.007,166.273,56.408,160.251
C06887=1015.881,61.147,-114.022,166.277,56.398,160.250
C06888=1015.886,61.396,-114.037,166.280,56.389,160.249
C06889=1015.891,61.646,-114.053,166.282,56.379,160.247
C06890=1015.896,61.895,-114.068,166.285,56.370,160.246
C06891=1015.902,62.145,-114.083,166.287,56.361,160.245
C06892=1015.907,62.394,-114.099,166.289,56.351,160.244
C06893=1015.911,62.644,-114.114,166.292,56.342,160.242
C06894=1015.916,62.893,-114.129,166.295,56.333,160.241
C06895=1015.922,63.143,-114.145,166.297,56.324,160.240
C06896=1015.926,63.393,-114.161,166.300,56.314,160.239
C06897=1015.931,63.642,-114.176,166.302,56.305,160.237
C06898=1015.937,63.892,-114.191,166.305,56.296,160.237
C06899=1015.941,64.141,-114.207,166.307,56.287,160.235
C06900=1015.946,64.391,-114.222,166.310,56.277,160.234
C06901=1015.952,64.639,-114.238,166.313,56.268,160.233
C06902=1015.956,64.890,-114.254,166.315,56.259,160.232
C06903=1015.961,65.139,-114.270,166.317,56.250,160.230
C06904=1015.966,65.388,-114.285,166.319,56.241,160.229
C06905=1015.971,65.638,-114.301,166.322,56.232,160.228
C06906=1015.977,65.887,-114.317,166.324,56.222,160.227
C06907=1015.981,66.137,-114.333,166.327,56.213,160.225
C06908=1015.986,66.386,-114.348,166.329,56.204,160.224
C06909=1015.991,66.636,-114.364,166.332,56.194,160.223
C06910=1015.996,66.885,-114.379,166.335,56.186,160.222
C06911=1016.001,67.134,-114.395,166.337,56.176,160.221
C06912=1016.006,67.384,-114.411,166.340,56.167,160.219
C06913=1016.011,67.634,-114.426,166.342,56.157,160.218
C06914=1016.016,67.883,-114.442,166.345,56.149,160.217
C06915=1016.022,68.133,-114.458,166.348,56.139,160.216
C06916=1016.026,68.382,-114.474,166.350,56.130,160.215
C06917=1016.031,68.631,-114.489,166.352,56.120,160.213
C06918=1016.036,68.880,-114.506,166.355,56.112,160.212
C06919=1016.041,69.130,-114.521,166.358,56.102,160.211
C06920=1016.046,69.379,-114.538,166.360,56.093,160.210
C06921=1016.051,69.629,-114.553,166.363,56.083,160.209
C06922=1016.056,69.879,-114.569,166.366,56.075,160.208
C06923=1016.060,70.128,-114.586,166.368,56.065,160.206
C06924=1016.066,70.378,-114.601,166.371,56.056,160.205
C06925=1016.070,70.627,-114.617,166.373,56.047,160.204
C06926=1016.076,70.876,-114.633,166.376,56.037,160.203
C06927=1016.081,71.126,-114.649,166.378,56.029,160.202
C06928=1016.086,71.375,-114.665,166.380,56.020,160.200
C06929=1016.090,71.624,-114.681,166.383,56.010,160.199
C06930=1016.095,71.874,-114.697,166.385,56.001,160.198
C06931=1016.101,72.123,-114.713,166.388,55.991,160.197
C06932=1016.105,72.372,-114.729,166.391,55.983,160.196
C06933=1016.111,72.622,-114.745,166.393,55.973,160.194
C06934=1016.115,72.872,-114.760,166.396,55.964,160.193
C06935=1016.120,73.122,-114.777,166.398,55.955,160.192
C06936=1016.125,73.371,-114.792,166.401,55.945,160.191
C06937=1016.130,73.620,-114.809,166.403,55.936,160.189
C06938=1016.136,73.870,-114.824,166.406,55.927,160.188
C06939=1016.140,74.119,-114.841,166.409,55.918,160.187
C06940=1016.146,74.400,-114.859,166.412,55.907,160.186
C06941=1016.152,74.682,-114.877,166.415,55.897,160.184
C06942=1016.158,74.962,-114.896,166.418,55.886,160.183
C06943=1016.163,75.244,-114.914,166.421,55.876,160.182
C06944=1016.168,75.493,-114.929,166.423,55.866,160.180
C06945=1016.173,75.743,-114.946,166.426,55.857,160.179
C06946=1016.177,75.992,-114.962,166.428,55.848,160.178
C06947=1016.183,76.242,-114.978,166.431,55.838,160.177
C06948=1016.188,76.491,-114.994,166.433,55.829,160.175
C06949=1016.192,76.740,-115.010,166.436,55.820,160.174
C06950=1016.198,76.990,-115.026,166.439,55.811,160.173
C06951=1016.203,77.239,-115.043,166.442,55.802,160.172
C06952=1016.208,77.489,-115.059,166.444,55.792,160.171
C06953=1016.212,77.738,-115.075,166.447,55.783,160.169
C06954=1016.217,77.987,-115.092,166.449,55.775,160.168
C06955=1016.222,78.237,-115.108,166.451,55.765,160.167
C06956=1016.227,78.487,-115.125,166.454,55.756,160.166
C06957=1016.232,78.736,-115.141,166.456,55.747,160.165
C06958=1016.237,78.985,-115.158,166.459,55.737,160.163
C06959=1016.242,79.235,-115.173,166.462,55.729,160.162
C06960=1016.247,79.484,-115.190,166.464,55.719,160.161
C06961=1016.252,79.733,-115.207,166.467,55.710,160.160
C06962=1016.256,79.982,-115.223,166.470,55.701,160.159
C06963=1016.261,80.232,-115.239,166.472,55.691,160.157
C06964=1016.266,80.481,-115.256,166.475,55.683,160.156
C06965=1016.271,80.731,-115.273,166.478,55.673,160.155
C06966=1016.276,80.980,-115.289,166.480,55.664,160.154
C06967=1016.281,81.230,-115.306,166.483,55.655,160.153
C06968=1016.286,81.479,-115.321,166.485,55.645,160.152
C06969=1016.291,81.729,-115.338,166.488,55.636,160.150
C06970=1016.296,81.978,-115.355,166.491,55.627,160.149
C06971=1016.301,82.227,-115.371,166.494,55.618,160.148
C06972=1016.306,82.477,-115.388,166.496,55.609,160.147
C06973=1016.310,82.726,-115.404,166.499,55.599,160.146
C06974=1016.316,82.976,-115.421,166.501,55.590,160.144
C06975=1016.320,83.225,-115.437,166.504,55.581,160.143
C06976=1016.325,83.475,-115.454,166.507,55.571,160.142
C06977=1016.330,83.724,-115.471,166.509,55.562,160.141
C06978=1016.336,83.973,-115.487,166.512,55.553,160.139
C06979=1016.341,84.222,-115.503,166.514,55.543,160.138
C06980=1016.345,84.472,-115.520,166.517,55.534,160.137
C06981=1016.350,84.721,-115.536,166.520,55.525,160.136
C06982=1016.355,84.971,-115.553,166.522,55.516,160.135
C06983=1016.361,85.221,-115.570,166.525,55.506,160.133
C06984=1016.365,85.470,-115.586,166.527,55.497,160.132
C06985=1016.370,85.719,-115.603,166.531,55.488,160.131
C06986=1016.375,85.968,-115.620,166.533,55.479,160.130
C06987=1016.380,86.218,-115.636,166.536,55.470,160.129
C06988=1016.385,86.467,-115.653,166.538,55.460,160.127
C06989=1016.390,86.717,-115.668,166.541,55.451,160.126
C06990=1016.396,86.966,-115.685,166.544,55.442,160.125
C06991=1016.400,87.215,-115.702,166.546,55.432,160.124
C06992=1016.405,87.465,-115.719,166.549,55.423,160.123
C06993=1016.410,87.714,-115.735,166.551,55.414,160.121
C06994=1016.415,87.964,-115.752,166.554,55.404,160.120
C06995=1016.421,88.213,-115.769,166.556,55.395,160.119
C06996=1016.425,88.462,-115.785,166.560,55.385,160.117
C06997=1016.430,88.712,-115.802,166.562,55.376,160.116
C06998=1016.436,88.962,-115.819,166.565,55.366,160.115
C06999=1016.440,89.211,-115.835,166.568,55.358,160.114
C07000=1016.445,89.460,-115.852,166.571,55.348,160.113
C07001=1016.450,89.710,-115.870,166.572,55.340,160.111
C07002=1016.454,89.959,-115.886,166.575,55.330,160.110
C07003=1016.460,90.208,-115.904,166.578,55.321,160.109
C07004=1016.465,90.490,-115.922,166.581,55.311,160.108
C07005=1016.471,90.771,-115.941,166.584,55.300,160.106
C07006=1016.476,91.052,-115.960,166.587,55.290,160.105
C07007=1016.482,91.333,-115.980,166.590,55.279,160.104
C07008=1016.487,91.583,-115.997,166.593,55.270,160.103
C07009=1016.491,91.832,-116.014,166.596,55.261,160.101
C07010=1016.497,92.081,-116.031,166.598,55.252,160.100
C07011=1016.502,92.331,-116.048,166.601,55.242,160.099
C07012=1016.506,92.580,-116.065,166.604,55.233,160.098
C07013=1016.511,92.830,-116.082,166.607,55.224,160.097
C07014=1016.516,93.080,-116.099,166.610,55.215,160.095
C07015=1016.521,93.328,-116.116,166.612,55.206,160.094
C07016=1016.526,93.578,-116.133,166.615,55.197,160.093
C07017=1016.531,93.828,-116.150,166.618,55.187,160.092
C07018=1016.535,94.077,-116.167,166.620,55.178,160.091
C07019=1016.541,94.326,-116.184,166.623,55.169,160.089
C07020=1016.546,94.575,-116.201,166.626,55.160,160.088
C07021=1016.550,94.825,-116.218,166.628,55.150,160.087
C07022=1016.555,95.074,-116.235,166.631,55.141,160.086
C07023=1016.561,95.323,-116.253,166.634,55.132,160.085
C07024=1016.566,95.573,-116.270,166.636,55.123,160.083
C07025=1016.570,95.822,-116.287,166.639,55.113,160.082
C07026=1016.575,96.072,-116.303,166.642,55.104,160.081
C07027=1016.581,96.321,-116.321,166.644,55.095,160.080
C07028=1016.586,96.571,-116.338,166.647,55.086,160.078
C07029=1016.590,96.820,-116.355,166.650,55.076,160.077
C07030=1016.595,97.069,-116.373,166.653,55.067,160.076
C07031=1016.600,97.318,-116.389,166.655,55.058,160.075
C07032=1016.605,97.567,-116.406,166.659,55.048,160.074
C07033=1016.611,97.816,-116.423,166.662,55.039,160.073
C07034=1016.615,98.066,-116.441,166.664,55.030,160.071
C07035=1016.620,98.316,-116.458,166.667,55.021,160.070
C07036=1016.626,98.565,-116.475,166.669,55.011,160.069
C07037=1016.630,98.814,-116.492,166.672,55.001,160.067
C07038=1016.635,99.064,-116.509,166.675,54.992,160.066
C07039=1016.640,99.313,-116.527,166.678,54.984,160.065
C07040=1016.645,99.563,-116.544,166.681,54.974,160.064
C07041=1016.650,99.811,-116.561,166.683,54.965,160.063
C07042=1016.654,100.061,-116.579,166.686,54.956,160.062
C07043=1016.660,100.310,-116.596,166.689,54.947,160.060
C07044=1016.664,100.560,-116.614,166.692,54.937,160.059
C07045=1016.670,100.809,-116.631,166.694,54.928,160.058
C07046=1016.674,101.059,-116.649,166.697,54.919,160.057
C07047=1016.679,101.308,-116.666,166.700,54.910,160.056
C07048=1016.684,101.557,-116.684,166.703,54.901,160.054
C07049=1016.688,101.807,-116.702,166.705,54.891,160.053
C07050=1016.694,102.056,-116.719,166.708,54.882,160.052
C07051=1016.698,102.305,-116.736,166.711,54.873,160.051
C07052=1016.703,102.554,-116.754,166.714,54.864,160.050
C07053=1016.708,102.804,-116.771,166.717,54.855,160.049
C07054=1016.713,103.053,-116.789,166.720,54.846,160.047
C07055=1016.718,103.303,-116.807,166.722,54.837,160.046
C07056=1016.723,103.552,-116.824,166.725,54.828,160.045
C07057=1016.728,103.801,-116.842,166.728,54.818,160.044
C07058=1016.733,104.051,-116.859,166.731,54.809,160.043
C07059=1016.737,104.300,-116.877,166.733,54.800,160.041
C07060=1016.743,104.549,-116.894,166.736,54.791,160.040
C07061=1016.747,104.799,-116.912,166.739,54.782,160.039
C07062=1016.752,105.048,-116.930,166.742,54.772,160.038
C07063=1016.757,105.297,-116.947,166.744,54.763,160.037
C07064=1016.762,105.547,-116.965,166.747,54.754,160.035
C07065=1016.767,105.796,-116.982,166.750,54.745,160.034
C07066=1016.772,106.045,-117.000,166.753,54.736,160.033
C07067=1016.777,106.295,-117.017,166.757,54.726,160.032
C07068=1016.782,106.577,-117.037,166.758,54.715,160.030
C07069=1016.789,106.858,-117.057,166.762,54.705,160.029
C07070=1016.794,107.139,-117.077,166.765,54.695,160.028
C07071=1016.799,107.421,-117.097,166.768,54.685,160.026
C07072=1016.804,107.670,-117.115,166.772,54.675,160.025
C07073=1016.809,107.920,-117.133,166.775,54.666,160.024
C07074=1016.815,108.169,-117.150,166.777,54.656,160.023
C07075=1016.819,108.419,-117.168,166.780,54.647,160.021
C07076=1016.824,108.667,-117.185,166.783,54.638,160.020
C07077=1016.829,108.916,-117.203,166.786,54.628,160.019
C07078=1016.834,109.166,-117.220,166.788,54.619,160.018
C07079=1016.839,109.415,-117.238,166.791,54.610,160.017
C07080=1016.844,109.665,-117.256,166.794,54.601,160.015
C07081=1016.849,109.914,-117.274,166.797,54.592,160.014
C07082=1016.854,110.163,-117.292,166.800,54.583,160.013
C07083=1016.859,110.412,-117.310,166.802,54.573,160.012
C07084=1016.863,110.662,-117.328,166.805,54.564,160.011
C07085=1016.869,110.911,-117.345,166.809,54.555,160.010
C07086=1016.874,111.161,-117.363,166.812,54.546,160.008
C07087=1016.878,111.410,-117.381,166.815,54.536,160.007
C07088=1016.883,111.659,-117.400,166.818,54.527,160.006
C07089=1016.889,111.909,-117.417,166.820,54.518,160.005
C07090=1016.893,112.158,-117.435,166.823,54.509,160.004
C07091=1016.898,112.407,-117.454,166.826,54.500,160.002
C07092=1016.903,112.657,-117.472,166.829,54.491,160.001
C07093=1016.908,112.906,-117.490,166.832,54.482,160.000
C07094=1016.912,113.155,-117.508,166.835,54.473,159.999
C07095=1016.917,113.404,-117.526,166.838,54.464,159.998
C07096=1016.922,113.653,-117.544,166.841,54.455,159.997
C07097=1016.926,113.903,-117.562,166.844,54.446,159.996
C07098=1016.931,114.152,-117.580,166.846,54.436,159.994
C07099=1016.936,114.401,-117.598,166.849,54.427,159.993
C07100=1016.941,114.651,-117.617,166.852,54.418,159.992
C07101=1016.945,114.900,-117.635,166.855,54.410,159.991
C07102=1016.951,115.149,-117.654,166.858,54.401,159.990
C07103=1016.955,115.398,-117.672,166.861,54.391,159.989
C07104=1016.959,115.648,-117.691,166.864,54.382,159.987
C07105=1016.964,115.897,-117.709,166.867,54.373,159.986
C07106=1016.969,116.146,-117.727,166.870,54.364,159.985
C07107=1016.974,116.396,-117.745,166.873,54.355,159.984
C07108=1016.978,116.645,-117.763,166.875,54.346,159.983
C07109=1016.983,116.895,-117.781,166.878,54.337,159.982
C07110=1016.988,117.143,-117.800,166.881,54.328,159.980
C07111=1016.993,117.393,-117.818,166.884,54.318,159.979
C07112=1016.998,117.642,-117.837,166.887,54.309,159.978
C07113=1017.003,117.891,-117.855,166.890,54.301,159.977
C07114=1017.008,118.141,-117.873,166.893,54.292,159.976
C07115=1017.013,118.390,-117.892,166.896,54.283,159.975
C07116=1017.018,118.639,-117.910,166.899,54.274,159.973
C07117=1017.023,118.889,-117.928,166.902,54.264,159.972
C07118=1017.027,119.138,-117.947,166.905,54.255,159.971
C07119=1017.032,119.387,-117.965,166.908,54.246,159.970
C07120=1017.037,119.636,-117.984,166.910,54.237,159.969
C07121=1017.042,119.886,-118.002,166.913,54.228,159.968
C07122=1017.047,120.135,-118.020,166.916,54.219,159.966
C07123=1017.052,120.384,-118.038,166.919,54.210,159.965
C07124=1017.056,120.634,-118.056,166.923,54.200,159.964
C07125=1017.062,120.882,-118.075,166.926,54.191,159.963
C07126=1017.066,121.132,-118.093,166.929,54.182,159.962
C07127=1017.071,121.381,-118.112,166.932,54.173,159.961
C07128=1017.077,121.630,-118.131,166.935,54.164,159.959
C07129=1017.082,121.880,-118.149,166.938,54.155,159.958
C07130=1017.086,122.129,-118.167,166.940,54.146,159.957
C07131=1017.091,122.379,-118.185,166.943,54.137,159.956
C07132=1017.096,122.660,-118.206,166.947,54.126,159.955
C07133=1017.102,122.942,-118.227,166.950,54.115,159.953
C07134=1017.107,123.223,-118.248,166.953,54.105,159.952
C07135=1017.113,123.504,-118.269,166.957,54.095,159.951
C07136=1017.118,123.754,-118.287,166.960,54.086,159.949
C07137=1017.123,124.003,-118.306,166.964,54.077,159.948
C07138=1017.128,124.253,-118.324,166.967,54.067,159.947
C07139=1017.133,124.502,-118.342,166.969,54.058,159.946
C07140=1017.138,124.751,-118.361,166.972,54.049,159.945
C07141=1017.143,125.000,-118.379,166.975,54.040,159.944
C07142=1017.149,125.249,-118.399,166.978,54.030,159.942
C07143=1017.153,125.499,-118.417,166.981,54.021,159.941
C07144=1017.157,125.748,-118.436,166.985,54.012,159.940
C07145=1017.162,125.997,-118.455,166.988,54.003,159.939
C07146=1017.167,126.246,-118.473,166.991,53.994,159.938
C07147=1017.172,126.496,-118.491,166.993,53.985,159.936
C07148=1017.178,126.745,-118.510,166.996,53.976,159.935
C07149=1017.182,126.995,-118.528,166.999,53.967,159.934
C07150=1017.188,127.243,-118.547,167.003,53.957,159.933
C07151=1017.192,127.493,-118.565,167.006,53.948,159.932
C07152=1017.197,127.742,-118.583,167.009,53.939,159.931
C07153=1017.203,127.991,-118.603,167.012,53.929,159.929
C07154=1017.208,128.241,-118.621,167.015,53.920,159.928
C07155=1017.213,128.490,-118.640,167.019,53.911,159.927
C07156=1017.217,128.739,-118.658,167.022,53.902,159.926
C07157=1017.223,128.988,-118.677,167.025,53.893,159.925
C07158=1017.228,129.238,-118.695,167.028,53.884,159.924
C07159=1017.233,129.486,-118.714,167.031,53.875,159.922
